LIN {X -0.145,Y -338.267,Z 1435.514,A 0.000,B 0.000,C 90.000,E1 272.579} C_DIS
LIN {X 0.126,Y -330.256,Z 1435.514,A 0.000,B 0.000,C 90.000,E1 272.407} C_DIS
LIN {X -0.143,Y -321.454,Z 1435.513,A 0.000,B 0.000,C 90.000,E1 272.350} C_DIS
LIN {X 0.117,Y -311.305,Z 1435.513,A 0.000,B 0.000,C 90.000,E1 272.236} C_DIS
LIN {X 0.012,Y -305.881,Z 1435.512,A 0.000,B 0.000,C 90.000,E1 272.236} C_DIS
LIN {X -0.024,Y -181.226,Z 1435.512,A 0.000,B 0.000,C 90.000,E1 272.236} C_DIS
LIN {X 0.021,Y -181.579,Z 1435.501,A 0.000,B 0.000,C 90.000,E1 270.172} C_DIS
LIN {X 0.010,Y -180.886,Z 1435.473,A 0.000,B 0.000,C 90.000,E1 265.122} C_DIS
LIN {X 0.070,Y -179.008,Z 1435.445,A 0.000,B 0.000,C 90.000,E1 260.038} C_DIS
LIN {X -0.012,Y -178.617,Z 1435.440,A 0.000,B 0.000,C 90.000,E1 259.218} C_DIS
LIN {X 0.056,Y -175.669,Z 1435.412,A 0.000,B 0.000,C 90.000,E1 254.102} C_DIS
LIN {X 0.061,Y -172.386,Z 1435.388,A 0.000,B 0.000,C 90.000,E1 249.826} C_DIS
LIN {X 0.075,Y -171.187,Z 1435.379,A 0.000,B 0.000,C 90.000,E1 248.103} C_DIS
LIN {X -0.032,Y -167.479,Z 1435.354,A 0.000,B 0.000,C 90.000,E1 243.819} C_DIS
LIN {X -0.025,Y -166.875,Z 1435.350,A 0.000,B 0.000,C 90.000,E1 242.948} C_DIS
LIN {X -0.032,Y -162.180,Z 1435.321,A 0.000,B 0.000,C 90.000,E1 237.709} C_DIS
LIN {X 0.025,Y -160.746,Z 1435.311,A 0.000,B 0.000,C 90.000,E1 235.928} C_DIS
LIN {X 0.003,Y -157.546,Z 1435.291,A 0.000,B 0.000,C 90.000,E1 232.396} C_DIS
LIN {X -0.058,Y -155.574,Z 1435.276,A 0.000,B 0.000,C 90.000,E1 229.747} C_DIS
LIN {X -0.006,Y -151.860,Z 1435.251,A 0.000,B 0.000,C 90.000,E1 225.243} C_DIS
LIN {X 0.007,Y -150.083,Z 1435.236,A 0.000,B 0.000,C 90.000,E1 222.528} C_DIS
LIN {X 0.041,Y -146.886,Z 1435.211,A 0.000,B 0.000,C 90.000,E1 217.971} C_DIS
LIN {X 0.030,Y -145.473,Z 1435.196,A 0.000,B 0.000,C 90.000,E1 215.231} C_DIS
LIN {X -0.053,Y -142.884,Z 1435.170,A 0.000,B 0.000,C 90.000,E1 210.669} C_DIS
LIN {X 0.004,Y -141.503,Z 1435.150,A 0.000,B 0.000,C 90.000,E1 206.950} C_DIS
LIN {X 0.053,Y -139.389,Z 1435.114,A 0.000,B 0.000,C 90.000,E1 200.429} C_DIS
LIN {X -0.027,Y -139.096,Z 1435.103,A 0.000,B 0.000,C 90.000,E1 198.598} C_DIS
LIN {X -0.035,Y -138.353,Z 1435.057,A 0.000,B 0.000,C 90.000,E1 190.197} C_DIS
LIN {X -0.043,Y -139.516,Z 1435.005,A 0.000,B 0.000,C 90.000,E1 180.859} C_DIS
LIN {X 0.038,Y -141.171,Z 1434.974,A 0.000,B 0.000,C 90.000,E1 175.241} C_DIS
LIN {X 0.009,Y -142.550,Z 1434.958,A 0.000,B 0.000,C 90.000,E1 172.470} C_DIS
LIN {X -0.065,Y -144.826,Z 1434.932,A 0.000,B 0.000,C 90.000,E1 167.881} C_DIS
LIN {X 0.063,Y -147.449,Z 1434.912,A 0.000,B 0.000,C 90.000,E1 164.157} C_DIS
LIN {X -0.050,Y -150.030,Z 1434.892,A 0.000,B 0.000,C 90.000,E1 160.550} C_DIS
LIN {X -0.044,Y -153.367,Z 1434.872,A 0.000,B 0.000,C 90.000,E1 156.922} C_DIS
LIN {X 0.005,Y -155.901,Z 1434.857,A 0.000,B 0.000,C 90.000,E1 154.204} C_DIS
LIN {X -0.019,Y -159.761,Z 1434.837,A 0.000,B 0.000,C 90.000,E1 150.639} C_DIS
LIN {X -0.032,Y -162.001,Z 1434.827,A 0.000,B 0.000,C 90.000,E1 148.869} C_DIS
LIN {X -0.013,Y -166.194,Z 1434.807,A 0.000,B 0.000,C 90.000,E1 145.341} C_DIS
LIN {X 0.085,Y -171.208,Z 1434.788,A 0.000,B 0.000,C 90.000,E1 141.823} C_DIS
LIN {X 0.009,Y -176.093,Z 1434.769,A 0.000,B 0.000,C 90.000,E1 138.405} C_DIS
LIN {X 0.000,Y -180.354,Z 1434.755,A 0.000,B 0.000,C 90.000,E1 135.850} C_DIS
LIN {X 0.104,Y -185.763,Z 1434.736,A 0.000,B 0.000,C 90.000,E1 132.447} C_DIS
LIN {X 0.037,Y -190.377,Z 1434.722,A 0.000,B 0.000,C 90.000,E1 129.967} C_DIS
LIN {X -0.063,Y -197.702,Z 1434.699,A 0.000,B 0.000,C 90.000,E1 125.884} C_DIS
LIN {X -0.012,Y -200.248,Z 1434.692,A 0.000,B 0.000,C 90.000,E1 124.612} C_DIS
LIN {X -0.078,Y -312.029,Z 1434.692,A 0.000,B 0.000,C 90.000,E1 124.612} C_DIS
LIN {X 0.044,Y -317.244,Z 1434.691,A 0.000,B 0.000,C 90.000,E1 124.405} C_DIS
LIN {X -0.034,Y -319.611,Z 1434.690,A 0.000,B 0.000,C 90.000,E1 124.246} C_DIS
LIN {X 0.116,Y -323.459,Z 1434.688,A 0.000,B 0.000,C 90.000,E1 123.785} C_DIS
LIN {X 0.010,Y -325.330,Z 1434.686,A 0.000,B 0.000,C 90.000,E1 123.499} C_DIS
LIN {X -0.099,Y -326.795,Z 1434.684,A 0.000,B 0.000,C 90.000,E1 123.214} C_DIS
LIN {X 0.023,Y -339.885,Z 1434.665,A 0.000,B 0.000,C 90.000,E1 119.745} C_DIS
LIN {X -0.091,Y -352.024,Z 1434.650,A 0.000,B 0.000,C 90.000,E1 117.001} C_DIS
LIN {X 0.137,Y -365.628,Z 1434.635,A 0.000,B 0.000,C 90.000,E1 114.259} C_DIS
LIN {X 0.193,Y -379.053,Z 1434.622,A 0.000,B 0.000,C 90.000,E1 111.897} C_DIS
LIN {X -0.052,Y -393.825,Z 1434.609,A 0.000,B 0.000,C 90.000,E1 109.631} C_DIS
LIN {X -0.205,Y -410.046,Z 1434.597,A 0.000,B 0.000,C 90.000,E1 107.402} C_DIS
LIN {X -0.078,Y -427.833,Z 1434.584,A 0.000,B 0.000,C 90.000,E1 105.190} C_DIS
LIN {X -0.073,Y -447.205,Z 1434.573,A 0.000,B 0.000,C 90.000,E1 103.063} C_DIS
LIN {X 0.056,Y -467.384,Z 1434.562,A 0.000,B 0.000,C 90.000,E1 101.074} C_DIS
LIN {X -0.132,Y -485.488,Z 1434.553,A 0.000,B 0.000,C 90.000,E1 99.500} C_DIS
LIN {X 0.022,Y -487.773,Z 1434.552,A 0.000,B 0.000,C 90.000,E1 99.265} C_DIS
LIN {X 0.176,Y -489.501,Z 1434.550,A 0.000,B 0.000,C 90.000,E1 99.029} C_DIS
LIN {X -0.002,Y -490.998,Z 1434.549,A 0.000,B 0.000,C 90.000,E1 98.803} C_DIS
LIN {X -0.103,Y -492.112,Z 1434.547,A 0.000,B 0.000,C 90.000,E1 98.568} C_DIS
LIN {X 0.124,Y -493.421,Z 1434.545,A 0.000,B 0.000,C 90.000,E1 98.049} C_DIS
LIN {X -0.129,Y -493.693,Z 1434.542,A 0.000,B 0.000,C 90.000,E1 97.587} C_DIS
LIN {X 0.117,Y -492.973,Z 1434.539,A 0.000,B 0.000,C 90.000,E1 97.068} C_DIS
LIN {X -0.125,Y -491.140,Z 1434.537,A 0.000,B 0.000,C 90.000,E1 96.606} C_DIS
LIN {X -0.221,Y -489.699,Z 1434.535,A 0.000,B 0.000,C 90.000,E1 96.372} C_DIS
LIN {X 0.050,Y -476.478,Z 1434.524,A 0.000,B 0.000,C 90.000,E1 94.359} C_DIS
LIN {X 0.126,Y -468.748,Z 1434.517,A 0.000,B 0.000,C 90.000,E1 93.094} C_DIS
LIN {X 0.040,Y -460.487,Z 1434.510,A 0.000,B 0.000,C 90.000,E1 91.835} C_DIS
LIN {X 0.052,Y -446.989,Z 1434.499,A 0.000,B 0.000,C 90.000,E1 89.771} C_DIS
LIN {X 0.071,Y -430.842,Z 1434.484,A 0.000,B 0.000,C 90.000,E1 87.135} C_DIS
LIN {X 0.169,Y -419.506,Z 1434.474,A 0.000,B 0.000,C 90.000,E1 85.241} C_DIS
LIN {X -0.006,Y -409.767,Z 1434.465,A 0.000,B 0.000,C 90.000,E1 83.628} C_DIS
LIN {X 0.192,Y -398.368,Z 1434.454,A 0.000,B 0.000,C 90.000,E1 81.659} C_DIS
LIN {X 0.153,Y -386.689,Z 1434.443,A 0.000,B 0.000,C 90.000,E1 79.690} C_DIS
LIN {X 0.023,Y -371.879,Z 1434.428,A 0.000,B 0.000,C 90.000,E1 77.117} C_DIS
LIN {X 0.103,Y -360.596,Z 1434.417,A 0.000,B 0.000,C 90.000,E1 75.046} C_DIS
LIN {X 0.006,Y -350.893,Z 1434.407,A 0.000,B 0.000,C 90.000,E1 73.268} C_DIS
LIN {X -0.058,Y -339.370,Z 1434.395,A 0.000,B 0.000,C 90.000,E1 71.148} C_DIS
LIN {X 0.075,Y -327.939,Z 1434.383,A 0.000,B 0.000,C 90.000,E1 68.954} C_DIS
LIN {X 0.059,Y -313.709,Z 1434.367,A 0.000,B 0.000,C 90.000,E1 66.102} C_DIS
LIN {X 0.019,Y -301.931,Z 1434.353,A 0.000,B 0.000,C 90.000,E1 63.512} C_DIS
LIN {X -0.058,Y -288.636,Z 1434.334,A 0.000,B 0.000,C 90.000,E1 60.205} C_DIS
LIN {X 0.031,Y -276.569,Z 1434.316,A 0.000,B 0.000,C 90.000,E1 56.786} C_DIS
LIN {X -0.168,Y -266.379,Z 1434.298,A 0.000,B 0.000,C 90.000,E1 53.703} C_DIS
LIN {X 0.058,Y -255.745,Z 1434.278,A 0.000,B 0.000,C 90.000,E1 50.114} C_DIS
LIN {X -0.098,Y -246.028,Z 1434.258,A 0.000,B 0.000,C 90.000,E1 46.539} C_DIS
LIN {X -0.060,Y -237.200,Z 1434.238,A 0.000,B 0.000,C 90.000,E1 42.852} C_DIS
LIN {X -0.091,Y -229.202,Z 1434.217,A 0.000,B 0.000,C 90.000,E1 39.116} C_DIS
LIN {X -0.089,Y -222.060,Z 1434.196,A 0.000,B 0.000,C 90.000,E1 35.311} C_DIS
LIN {X 0.043,Y -215.774,Z 1434.175,A 0.000,B 0.000,C 90.000,E1 31.416} C_DIS
LIN {X 0.010,Y -210.245,Z 1434.153,A 0.000,B 0.000,C 90.000,E1 27.513} C_DIS
LIN {X -0.029,Y -205.570,Z 1434.131,A 0.000,B 0.000,C 90.000,E1 23.567} C_DIS
LIN {X -0.066,Y -201.069,Z 1434.104,A 0.000,B 0.000,C 90.000,E1 18.779} C_DIS
LIN {X -0.076,Y -197.698,Z 1434.077,A 0.000,B 0.000,C 90.000,E1 13.939} C_DIS
LIN {X 0.037,Y -195.219,Z 1434.050,A 0.000,B 0.000,C 90.000,E1 9.029} C_DIS
LIN {X 0.028,Y -193.585,Z 1434.023,A 0.000,B 0.000,C 90.000,E1 4.131} C_DIS
LIN {X 0.095,Y -192.597,Z 1433.993,A 0.000,B 0.000,C 90.000,E1 358.682} C_DIS
LIN {X -0.049,Y -192.475,Z 1433.965,A 0.000,B 0.000,C 90.000,E1 353.799} C_DIS
LIN {X -0.037,Y -193.142,Z 1433.934,A 0.000,B 0.000,C 90.000,E1 348.049} C_DIS
LIN {X -0.074,Y -195.715,Z 1433.897,A 0.000,B 0.000,C 90.000,E1 341.511} C_DIS
LIN {X -0.024,Y -199.234,Z 1433.870,A 0.000,B 0.000,C 90.000,E1 336.613} C_DIS
LIN {X 0.017,Y -203.361,Z 1433.848,A 0.000,B 0.000,C 90.000,E1 332.564} C_DIS
LIN {X -0.051,Y -208.601,Z 1433.825,A 0.000,B 0.000,C 90.000,E1 328.584} C_DIS
LIN {X 0.060,Y -213.728,Z 1433.808,A 0.000,B 0.000,C 90.000,E1 325.388} C_DIS
LIN {X 0.014,Y -219.879,Z 1433.790,A 0.000,B 0.000,C 90.000,E1 322.271} C_DIS
LIN {X 0.041,Y -226.992,Z 1433.773,A 0.000,B 0.000,C 90.000,E1 319.175} C_DIS
LIN {X 0.005,Y -236.100,Z 1433.754,A 0.000,B 0.000,C 90.000,E1 315.769} C_DIS
LIN {X 0.090,Y -245.170,Z 1433.738,A 0.000,B 0.000,C 90.000,E1 312.771} C_DIS
LIN {X 0.108,Y -256.587,Z 1433.719,A 0.000,B 0.000,C 90.000,E1 309.483} C_DIS
LIN {X -0.062,Y -267.968,Z 1433.704,A 0.000,B 0.000,C 90.000,E1 306.664} C_DIS
LIN {X 0.025,Y -279.257,Z 1433.690,A 0.000,B 0.000,C 90.000,E1 304.199} C_DIS
LIN {X -0.015,Y -286.345,Z 1433.682,A 0.000,B 0.000,C 90.000,E1 302.832} C_DIS
LIN {X 0.036,Y -294.207,Z 1433.675,A 0.000,B 0.000,C 90.000,E1 301.465} C_DIS
LIN {X 0.043,Y -304.988,Z 1433.666,A 0.000,B 0.000,C 90.000,E1 299.795} C_DIS
LIN {X 0.023,Y -314.696,Z 1433.658,A 0.000,B 0.000,C 90.000,E1 298.487} C_DIS
LIN {X 0.044,Y -327.610,Z 1433.650,A 0.000,B 0.000,C 90.000,E1 296.950} C_DIS
LIN {X -0.026,Y -349.254,Z 1433.637,A 0.000,B 0.000,C 90.000,E1 294.695} C_DIS
LIN {X -0.169,Y -362.739,Z 1433.630,A 0.000,B 0.000,C 90.000,E1 293.334} C_DIS
LIN {X -0.059,Y -373.323,Z 1433.623,A 0.000,B 0.000,C 90.000,E1 292.206} C_DIS
LIN {X -0.032,Y -386.257,Z 1433.615,A 0.000,B 0.000,C 90.000,E1 290.791} C_DIS
LIN {X 0.149,Y -396.447,Z 1433.609,A 0.000,B 0.000,C 90.000,E1 289.631} C_DIS
LIN {X 0.159,Y -411.444,Z 1433.600,A 0.000,B 0.000,C 90.000,E1 287.946} C_DIS
LIN {X -0.072,Y -418.826,Z 1433.595,A 0.000,B 0.000,C 90.000,E1 287.149} C_DIS
LIN {X 0.042,Y -425.619,Z 1433.591,A 0.000,B 0.000,C 90.000,E1 286.315} C_DIS
LIN {X -0.062,Y -429.691,Z 1433.588,A 0.000,B 0.000,C 90.000,E1 285.788} C_DIS
LIN {X -0.023,Y -433.376,Z 1433.585,A 0.000,B 0.000,C 90.000,E1 285.245} C_DIS
LIN {X 0.114,Y -438.048,Z 1433.580,A 0.000,B 0.000,C 90.000,E1 284.426} C_DIS
LIN {X -0.015,Y -441.908,Z 1433.576,A 0.000,B 0.000,C 90.000,E1 283.647} C_DIS
LIN {X 0.210,Y -445.060,Z 1433.571,A 0.000,B 0.000,C 90.000,E1 282.827} C_DIS
LIN {X -0.207,Y -446.761,Z 1433.568,A 0.000,B 0.000,C 90.000,E1 282.355} C_DIS
LIN {X -0.178,Y -448.130,Z 1433.566,A 0.000,B 0.000,C 90.000,E1 281.827} C_DIS
LIN {X -0.141,Y -449.139,Z 1433.563,A 0.000,B 0.000,C 90.000,E1 281.299} C_DIS
LIN {X -0.180,Y -449.709,Z 1433.560,A 0.000,B 0.000,C 90.000,E1 280.782} C_DIS
LIN {X -0.128,Y -449.834,Z 1433.557,A 0.000,B 0.000,C 90.000,E1 280.254} C_DIS
LIN {X -0.076,Y -449.495,Z 1433.554,A 0.000,B 0.000,C 90.000,E1 279.726} C_DIS
LIN {X -0.098,Y -448.642,Z 1433.551,A 0.000,B 0.000,C 90.000,E1 279.208} C_DIS
LIN {X -0.050,Y -447.164,Z 1433.548,A 0.000,B 0.000,C 90.000,E1 278.681} C_DIS
LIN {X -0.077,Y -445.065,Z 1433.545,A 0.000,B 0.000,C 90.000,E1 278.163} C_DIS
LIN {X 0.157,Y -443.775,Z 1433.544,A 0.000,B 0.000,C 90.000,E1 277.871} C_DIS
LIN {X 0.113,Y -440.529,Z 1433.541,A 0.000,B 0.000,C 90.000,E1 277.352} C_DIS
LIN {X -0.158,Y -438.557,Z 1433.539,A 0.000,B 0.000,C 90.000,E1 277.125} C_DIS
LIN {X -0.223,Y -433.757,Z 1433.536,A 0.000,B 0.000,C 90.000,E1 276.606} C_DIS
LIN {X 0.144,Y -427.709,Z 1433.534,A 0.000,B 0.000,C 90.000,E1 276.030} C_DIS
LIN {X -0.192,Y -421.451,Z 1433.531,A 0.000,B 0.000,C 90.000,E1 275.625} C_DIS
LIN {X -0.102,Y -414.920,Z 1433.529,A 0.000,B 0.000,C 90.000,E1 275.220} C_DIS
LIN {X 0.100,Y -405.272,Z 1433.526,A 0.000,B 0.000,C 90.000,E1 274.702} C_DIS
LIN {X 0.072,Y -398.765,Z 1433.525,A 0.000,B 0.000,C 90.000,E1 274.416} C_DIS
LIN {X 0.148,Y -385.981,Z 1433.522,A 0.000,B 0.000,C 90.000,E1 273.898} C_DIS
LIN {X 0.082,Y -373.099,Z 1433.519,A 0.000,B 0.000,C 90.000,E1 273.440} C_DIS
LIN {X -0.154,Y -363.120,Z 1433.517,A 0.000,B 0.000,C 90.000,E1 273.151} C_DIS
LIN {X 0.060,Y -356.360,Z 1433.516,A 0.000,B 0.000,C 90.000,E1 272.922} C_DIS
LIN {X -0.102,Y -345.391,Z 1433.515,A 0.000,B 0.000,C 90.000,E1 272.694} C_DIS
LIN {X 0.077,Y -338.067,Z 1433.514,A 0.000,B 0.000,C 90.000,E1 272.522} C_DIS
LIN {X 0.032,Y -329.934,Z 1433.513,A 0.000,B 0.000,C 90.000,E1 272.407} C_DIS
LIN {X -0.033,Y -317.499,Z 1433.513,A 0.000,B 0.000,C 90.000,E1 272.293} C_DIS
LIN {X 0.007,Y -306.470,Z 1433.512,A 0.000,B 0.000,C 90.000,E1 272.236} C_DIS
LIN {X -0.024,Y -181.226,Z 1433.512,A 0.000,B 0.000,C 90.000,E1 272.236} C_DIS
LIN {X -0.023,Y -181.564,Z 1433.503,A 0.000,B 0.000,C 90.000,E1 270.516} C_DIS
LIN {X -0.034,Y -181.121,Z 1433.489,A 0.000,B 0.000,C 90.000,E1 267.993} C_DIS
LIN {X -0.045,Y -180.907,Z 1433.475,A 0.000,B 0.000,C 90.000,E1 265.469} C_DIS
LIN {X 0.012,Y -180.730,Z 1433.470,A 0.000,B 0.000,C 90.000,E1 264.609} C_DIS
LIN {X -0.066,Y -178.819,Z 1433.442,A 0.000,B 0.000,C 90.000,E1 259.567} C_DIS
LIN {X 0.015,Y -175.864,Z 1433.414,A 0.000,B 0.000,C 90.000,E1 254.448} C_DIS
LIN {X 0.064,Y -173.831,Z 1433.399,A 0.000,B 0.000,C 90.000,E1 251.873} C_DIS
LIN {X -0.001,Y -171.499,Z 1433.380,A 0.000,B 0.000,C 90.000,E1 248.465} C_DIS
LIN {X -0.014,Y -167.727,Z 1433.356,A 0.000,B 0.000,C 90.000,E1 244.152} C_DIS
LIN {X 0.002,Y -166.422,Z 1433.347,A 0.000,B 0.000,C 90.000,E1 242.410} C_DIS
LIN {X 0.000,Y -163.143,Z 1433.327,A 0.000,B 0.000,C 90.000,E1 238.918} C_DIS
LIN {X -0.034,Y -161.098,Z 1433.313,A 0.000,B 0.000,C 90.000,E1 236.294} C_DIS
LIN {X -0.050,Y -157.826,Z 1433.293,A 0.000,B 0.000,C 90.000,E1 232.763} C_DIS
LIN {X 0.013,Y -155.860,Z 1433.278,A 0.000,B 0.000,C 90.000,E1 230.070} C_DIS
LIN {X 0.069,Y -152.109,Z 1433.253,A 0.000,B 0.000,C 90.000,E1 225.567} C_DIS
LIN {X -0.024,Y -150.360,Z 1433.238,A 0.000,B 0.000,C 90.000,E1 222.894} C_DIS
LIN {X 0.016,Y -147.095,Z 1433.213,A 0.000,B 0.000,C 90.000,E1 218.338} C_DIS
LIN {X 0.011,Y -145.665,Z 1433.198,A 0.000,B 0.000,C 90.000,E1 215.598} C_DIS
LIN {X 0.013,Y -143.048,Z 1433.172,A 0.000,B 0.000,C 90.000,E1 211.003} C_DIS
LIN {X 0.014,Y -141.671,Z 1433.152,A 0.000,B 0.000,C 90.000,E1 207.308} C_DIS
LIN {X 0.058,Y -139.452,Z 1433.116,A 0.000,B 0.000,C 90.000,E1 200.791} C_DIS
LIN {X -0.021,Y -139.186,Z 1433.105,A 0.000,B 0.000,C 90.000,E1 198.960} C_DIS
LIN {X 0.002,Y -138.322,Z 1433.053,A 0.000,B 0.000,C 90.000,E1 189.613} C_DIS
LIN {X 0.009,Y -139.460,Z 1433.007,A 0.000,B 0.000,C 90.000,E1 181.203} C_DIS
LIN {X -0.051,Y -141.016,Z 1432.976,A 0.000,B 0.000,C 90.000,E1 175.641} C_DIS
LIN {X 0.040,Y -142.770,Z 1432.955,A 0.000,B 0.000,C 90.000,E1 171.894} C_DIS
LIN {X -0.005,Y -145.180,Z 1432.929,A 0.000,B 0.000,C 90.000,E1 167.297} C_DIS
LIN {X 0.028,Y -147.802,Z 1432.909,A 0.000,B 0.000,C 90.000,E1 163.614} C_DIS
LIN {X -0.077,Y -150.488,Z 1432.889,A 0.000,B 0.000,C 90.000,E1 160.007} C_DIS
LIN {X -0.004,Y -153.943,Z 1432.869,A 0.000,B 0.000,C 90.000,E1 156.357} C_DIS
LIN {X 0.059,Y -157.354,Z 1432.849,A 0.000,B 0.000,C 90.000,E1 152.743} C_DIS
LIN {X 0.003,Y -161.551,Z 1432.829,A 0.000,B 0.000,C 90.000,E1 149.203} C_DIS
LIN {X 0.014,Y -165.749,Z 1432.809,A 0.000,B 0.000,C 90.000,E1 145.674} C_DIS
LIN {X 0.002,Y -170.703,Z 1432.790,A 0.000,B 0.000,C 90.000,E1 142.190} C_DIS
LIN {X -0.087,Y -175.576,Z 1432.771,A 0.000,B 0.000,C 90.000,E1 138.771} C_DIS
LIN {X 0.032,Y -181.194,Z 1432.752,A 0.000,B 0.000,C 90.000,E1 135.324} C_DIS
LIN {X 0.026,Y -186.655,Z 1432.733,A 0.000,B 0.000,C 90.000,E1 131.962} C_DIS
LIN {X -0.030,Y -191.260,Z 1432.719,A 0.000,B 0.000,C 90.000,E1 129.483} C_DIS
LIN {X 0.050,Y -197.081,Z 1432.701,A 0.000,B 0.000,C 90.000,E1 126.171} C_DIS
LIN {X 0.063,Y -200.204,Z 1432.692,A 0.000,B 0.000,C 90.000,E1 124.612} C_DIS
LIN {X 0.063,Y -311.776,Z 1432.692,A 0.000,B 0.000,C 90.000,E1 124.612} C_DIS
LIN {X 0.137,Y -314.663,Z 1432.692,A 0.000,B 0.000,C 90.000,E1 124.532} C_DIS
LIN {X -0.170,Y -318.101,Z 1432.691,A 0.000,B 0.000,C 90.000,E1 124.405} C_DIS
LIN {X 0.050,Y -321.655,Z 1432.689,A 0.000,B 0.000,C 90.000,E1 124.040} C_DIS
LIN {X 0.153,Y -325.220,Z 1432.686,A 0.000,B 0.000,C 90.000,E1 123.499} C_DIS
LIN {X -0.032,Y -326.743,Z 1432.684,A 0.000,B 0.000,C 90.000,E1 123.214} C_DIS
LIN {X 0.079,Y -339.825,Z 1432.665,A 0.000,B 0.000,C 90.000,E1 119.745} C_DIS
LIN {X -0.030,Y -351.955,Z 1432.650,A 0.000,B 0.000,C 90.000,E1 117.001} C_DIS
LIN {X 0.042,Y -365.558,Z 1432.635,A 0.000,B 0.000,C 90.000,E1 114.283} C_DIS
LIN {X -0.102,Y -378.978,Z 1432.622,A 0.000,B 0.000,C 90.000,E1 111.950} C_DIS
LIN {X 0.003,Y -393.744,Z 1432.609,A 0.000,B 0.000,C 90.000,E1 109.631} C_DIS
LIN {X -0.149,Y -409.961,Z 1432.597,A 0.000,B 0.000,C 90.000,E1 107.402} C_DIS
LIN {X -0.022,Y -427.741,Z 1432.584,A 0.000,B 0.000,C 90.000,E1 105.190} C_DIS
LIN {X -0.029,Y -447.125,Z 1432.573,A 0.000,B 0.000,C 90.000,E1 103.063} C_DIS
LIN {X 0.097,Y -467.302,Z 1432.562,A 0.000,B 0.000,C 90.000,E1 101.074} C_DIS
LIN {X -0.073,Y -485.377,Z 1432.553,A 0.000,B 0.000,C 90.000,E1 99.500} C_DIS
LIN {X 0.060,Y -487.677,Z 1432.552,A 0.000,B 0.000,C 90.000,E1 99.265} C_DIS
LIN {X 0.043,Y -489.534,Z 1432.550,A 0.000,B 0.000,C 90.000,E1 99.029} C_DIS
LIN {X -0.049,Y -490.939,Z 1432.549,A 0.000,B 0.000,C 90.000,E1 98.803} C_DIS
LIN {X 0.242,Y -492.810,Z 1432.546,A 0.000,B 0.000,C 90.000,E1 98.276} C_DIS
LIN {X -0.019,Y -493.556,Z 1432.543,A 0.000,B 0.000,C 90.000,E1 97.814} C_DIS
LIN {X 0.219,Y -493.308,Z 1432.541,A 0.000,B 0.000,C 90.000,E1 97.296} C_DIS
LIN {X -0.027,Y -492.029,Z 1432.538,A 0.000,B 0.000,C 90.000,E1 96.834} C_DIS
LIN {X -0.178,Y -490.940,Z 1432.537,A 0.000,B 0.000,C 90.000,E1 96.606} C_DIS
LIN {X 0.060,Y -487.770,Z 1432.534,A 0.000,B 0.000,C 90.000,E1 96.087} C_DIS
LIN {X -0.006,Y -476.274,Z 1432.524,A 0.000,B 0.000,C 90.000,E1 94.359} C_DIS
LIN {X 0.065,Y -468.519,Z 1432.517,A 0.000,B 0.000,C 90.000,E1 93.094} C_DIS
LIN {X -0.020,Y -460.231,Z 1432.510,A 0.000,B 0.000,C 90.000,E1 91.835} C_DIS
LIN {X -0.011,Y -446.743,Z 1432.499,A 0.000,B 0.000,C 90.000,E1 89.771} C_DIS
LIN {X 0.004,Y -430.684,Z 1432.484,A 0.000,B 0.000,C 90.000,E1 87.135} C_DIS
LIN {X 0.095,Y -419.356,Z 1432.474,A 0.000,B 0.000,C 90.000,E1 85.241} C_DIS
LIN {X -0.080,Y -409.634,Z 1432.464,A 0.000,B 0.000,C 90.000,E1 83.628} C_DIS
LIN {X 0.122,Y -398.275,Z 1432.454,A 0.000,B 0.000,C 90.000,E1 81.659} C_DIS
LIN {X 0.078,Y -386.602,Z 1432.443,A 0.000,B 0.000,C 90.000,E1 79.690} C_DIS
LIN {X -0.055,Y -373.439,Z 1432.430,A 0.000,B 0.000,C 90.000,E1 77.409} C_DIS
LIN {X 0.063,Y -362.148,Z 1432.419,A 0.000,B 0.000,C 90.000,E1 75.338} C_DIS
LIN {X -0.002,Y -352.446,Z 1432.409,A 0.000,B 0.000,C 90.000,E1 73.559} C_DIS
LIN {X -0.146,Y -342.594,Z 1432.399,A 0.000,B 0.000,C 90.000,E1 71.764} C_DIS
LIN {X 0.049,Y -331.119,Z 1432.387,A 0.000,B 0.000,C 90.000,E1 69.571} C_DIS
LIN {X -0.001,Y -316.706,Z 1432.371,A 0.000,B 0.000,C 90.000,E1 66.741} C_DIS
LIN {X 0.058,Y -303.244,Z 1432.355,A 0.000,B 0.000,C 90.000,E1 63.819} C_DIS
LIN {X 0.027,Y -289.813,Z 1432.336,A 0.000,B 0.000,C 90.000,E1 60.511} C_DIS
LIN {X 0.012,Y -277.679,Z 1432.317,A 0.000,B 0.000,C 90.000,E1 57.120} C_DIS
LIN {X 0.064,Y -267.490,Z 1432.300,A 0.000,B 0.000,C 90.000,E1 53.989} C_DIS
LIN {X -0.053,Y -256.772,Z 1432.280,A 0.000,B 0.000,C 90.000,E1 50.481} C_DIS
LIN {X 0.012,Y -247.002,Z 1432.260,A 0.000,B 0.000,C 90.000,E1 46.863} C_DIS
LIN {X 0.076,Y -238.115,Z 1432.240,A 0.000,B 0.000,C 90.000,E1 43.176} C_DIS
LIN {X 0.074,Y -230.059,Z 1432.219,A 0.000,B 0.000,C 90.000,E1 39.439} C_DIS
LIN {X 0.055,Y -222.842,Z 1432.198,A 0.000,B 0.000,C 90.000,E1 35.644} C_DIS
LIN {X 0.018,Y -216.498,Z 1432.177,A 0.000,B 0.000,C 90.000,E1 31.799} C_DIS
LIN {X 0.003,Y -210.891,Z 1432.155,A 0.000,B 0.000,C 90.000,E1 27.897} C_DIS
LIN {X -0.015,Y -206.166,Z 1432.133,A 0.000,B 0.000,C 90.000,E1 23.951} C_DIS
LIN {X 0.046,Y -201.622,Z 1432.106,A 0.000,B 0.000,C 90.000,E1 19.141} C_DIS
LIN {X 0.057,Y -198.187,Z 1432.080,A 0.000,B 0.000,C 90.000,E1 14.300} C_DIS
LIN {X 0.021,Y -195.344,Z 1432.048,A 0.000,B 0.000,C 90.000,E1 8.624} C_DIS
LIN {X 0.061,Y -194.008,Z 1432.025,A 0.000,B 0.000,C 90.000,E1 4.531} C_DIS
LIN {X -0.035,Y -192.978,Z 1431.997,A 0.000,B 0.000,C 90.000,E1 359.542} C_DIS
LIN {X -0.037,Y -192.761,Z 1431.965,A 0.000,B 0.000,C 90.000,E1 353.799} C_DIS
LIN {X -0.014,Y -193.412,Z 1431.934,A 0.000,B 0.000,C 90.000,E1 348.049} C_DIS
LIN {X -0.038,Y -195.940,Z 1431.897,A 0.000,B 0.000,C 90.000,E1 341.511} C_DIS
LIN {X 0.021,Y -199.430,Z 1431.870,A 0.000,B 0.000,C 90.000,E1 336.613} C_DIS
LIN {X -0.111,Y -203.566,Z 1431.848,A 0.000,B 0.000,C 90.000,E1 332.615} C_DIS
LIN {X 0.009,Y -208.787,Z 1431.825,A 0.000,B 0.000,C 90.000,E1 328.584} C_DIS
LIN {X 0.127,Y -213.917,Z 1431.808,A 0.000,B 0.000,C 90.000,E1 325.388} C_DIS
LIN {X 0.086,Y -220.063,Z 1431.791,A 0.000,B 0.000,C 90.000,E1 322.271} C_DIS
LIN {X -0.051,Y -227.163,Z 1431.773,A 0.000,B 0.000,C 90.000,E1 319.218} C_DIS
LIN {X -0.082,Y -236.262,Z 1431.754,A 0.000,B 0.000,C 90.000,E1 315.810} C_DIS
LIN {X -0.013,Y -246.529,Z 1431.736,A 0.000,B 0.000,C 90.000,E1 312.447} C_DIS
LIN {X -0.126,Y -258.086,Z 1431.718,A 0.000,B 0.000,C 90.000,E1 309.197} C_DIS
LIN {X 0.113,Y -269.596,Z 1431.702,A 0.000,B 0.000,C 90.000,E1 306.297} C_DIS
LIN {X 0.079,Y -281.049,Z 1431.688,A 0.000,B 0.000,C 90.000,E1 303.865} C_DIS
LIN {X 0.066,Y -288.301,Z 1431.681,A 0.000,B 0.000,C 90.000,E1 302.498} C_DIS
LIN {X 0.144,Y -300.572,Z 1431.669,A 0.000,B 0.000,C 90.000,E1 300.463} C_DIS
LIN {X 0.072,Y -309.738,Z 1431.662,A 0.000,B 0.000,C 90.000,E1 299.155} C_DIS
LIN {X -0.137,Y -322.067,Z 1431.653,A 0.000,B 0.000,C 90.000,E1 297.641} C_DIS
LIN {X 0.065,Y -332.776,Z 1431.647,A 0.000,B 0.000,C 90.000,E1 296.411} C_DIS
LIN {X -0.075,Y -351.818,Z 1431.636,A 0.000,B 0.000,C 90.000,E1 294.463} C_DIS
LIN {X -0.057,Y -365.223,Z 1431.628,A 0.000,B 0.000,C 90.000,E1 293.078} C_DIS
LIN {X -0.109,Y -375.716,Z 1431.622,A 0.000,B 0.000,C 90.000,E1 291.972} C_DIS
LIN {X -0.127,Y -388.630,Z 1431.614,A 0.000,B 0.000,C 90.000,E1 290.556} C_DIS
LIN {X -0.086,Y -401.158,Z 1431.606,A 0.000,B 0.000,C 90.000,E1 289.141} C_DIS
LIN {X 0.044,Y -416.135,Z 1431.597,A 0.000,B 0.000,C 90.000,E1 287.457} C_DIS
LIN {X 0.130,Y -423.196,Z 1431.592,A 0.000,B 0.000,C 90.000,E1 286.622} C_DIS
LIN {X -0.120,Y -429.517,Z 1431.588,A 0.000,B 0.000,C 90.000,E1 285.843} C_DIS
LIN {X 0.091,Y -434.908,Z 1431.583,A 0.000,B 0.000,C 90.000,E1 285.009} C_DIS
LIN {X -0.174,Y -439.369,Z 1431.579,A 0.000,B 0.000,C 90.000,E1 284.245} C_DIS
LIN {X 0.129,Y -443.030,Z 1431.575,A 0.000,B 0.000,C 90.000,E1 283.411} C_DIS
LIN {X 0.141,Y -445.110,Z 1431.572,A 0.000,B 0.000,C 90.000,E1 282.883} C_DIS
LIN {X 0.164,Y -446.862,Z 1431.569,A 0.000,B 0.000,C 90.000,E1 282.355} C_DIS
LIN {X 0.194,Y -448.267,Z 1431.566,A 0.000,B 0.000,C 90.000,E1 281.827} C_DIS
LIN {X 0.234,Y -449.307,Z 1431.563,A 0.000,B 0.000,C 90.000,E1 281.299} C_DIS
LIN {X 0.195,Y -449.969,Z 1431.560,A 0.000,B 0.000,C 90.000,E1 280.782} C_DIS
LIN {X -0.194,Y -450.157,Z 1431.557,A 0.000,B 0.000,C 90.000,E1 280.310} C_DIS
LIN {X -0.141,Y -449.856,Z 1431.554,A 0.000,B 0.000,C 90.000,E1 279.782} C_DIS
LIN {X -0.162,Y -449.053,Z 1431.551,A 0.000,B 0.000,C 90.000,E1 279.265} C_DIS
LIN {X -0.181,Y -447.686,Z 1431.548,A 0.000,B 0.000,C 90.000,E1 278.746} C_DIS
LIN {X -0.138,Y -445.684,Z 1431.546,A 0.000,B 0.000,C 90.000,E1 278.219} C_DIS
LIN {X -0.167,Y -442.963,Z 1431.543,A 0.000,B 0.000,C 90.000,E1 277.701} C_DIS
LIN {X -0.212,Y -439.362,Z 1431.540,A 0.000,B 0.000,C 90.000,E1 277.182} C_DIS
LIN {X 0.001,Y -437.226,Z 1431.538,A 0.000,B 0.000,C 90.000,E1 276.891} C_DIS
LIN {X -0.073,Y -431.995,Z 1431.535,A 0.000,B 0.000,C 90.000,E1 276.372} C_DIS
LIN {X 0.113,Y -425.941,Z 1431.533,A 0.000,B 0.000,C 90.000,E1 275.853} C_DIS
LIN {X -0.103,Y -419.637,Z 1431.530,A 0.000,B 0.000,C 90.000,E1 275.454} C_DIS
LIN {X 0.145,Y -413.144,Z 1431.528,A 0.000,B 0.000,C 90.000,E1 275.049} C_DIS
LIN {X 0.003,Y -403.235,Z 1431.526,A 0.000,B 0.000,C 90.000,E1 274.588} C_DIS
LIN {X -0.041,Y -393.561,Z 1431.523,A 0.000,B 0.000,C 90.000,E1 274.188} C_DIS
LIN {X 0.173,Y -380.809,Z 1431.521,A 0.000,B 0.000,C 90.000,E1 273.669} C_DIS
LIN {X -0.168,Y -367.765,Z 1431.518,A 0.000,B 0.000,C 90.000,E1 273.269} C_DIS
LIN {X 0.089,Y -357.480,Z 1431.516,A 0.000,B 0.000,C 90.000,E1 272.922} C_DIS
LIN {X -0.099,Y -346.344,Z 1431.515,A 0.000,B 0.000,C 90.000,E1 272.694} C_DIS
LIN {X 0.072,Y -339.001,Z 1431.514,A 0.000,B 0.000,C 90.000,E1 272.522} C_DIS
LIN {X 0.049,Y -326.341,Z 1431.513,A 0.000,B 0.000,C 90.000,E1 272.350} C_DIS
LIN {X 0.152,Y -314.275,Z 1431.513,A 0.000,B 0.000,C 90.000,E1 272.236} C_DIS
LIN {X 0.005,Y -307.328,Z 1431.512,A 0.000,B 0.000,C 90.000,E1 272.236} C_DIS
LIN {X -0.025,Y -181.226,Z 1431.512,A 0.000,B 0.000,C 90.000,E1 272.236} C_DIS
LIN {X -0.026,Y -181.564,Z 1431.503,A 0.000,B 0.000,C 90.000,E1 270.516} C_DIS
LIN {X -0.036,Y -181.121,Z 1431.489,A 0.000,B 0.000,C 90.000,E1 267.993} C_DIS
LIN {X -0.047,Y -180.907,Z 1431.475,A 0.000,B 0.000,C 90.000,E1 265.469} C_DIS
LIN {X 0.009,Y -180.730,Z 1431.470,A 0.000,B 0.000,C 90.000,E1 264.609} C_DIS
LIN {X -0.070,Y -178.819,Z 1431.442,A 0.000,B 0.000,C 90.000,E1 259.567} C_DIS
LIN {X 0.013,Y -175.863,Z 1431.414,A 0.000,B 0.000,C 90.000,E1 254.448} C_DIS
LIN {X 0.062,Y -173.831,Z 1431.399,A 0.000,B 0.000,C 90.000,E1 251.873} C_DIS
LIN {X -0.003,Y -171.498,Z 1431.380,A 0.000,B 0.000,C 90.000,E1 248.465} C_DIS
LIN {X -0.017,Y -167.726,Z 1431.356,A 0.000,B 0.000,C 90.000,E1 244.152} C_DIS
LIN {X 0.000,Y -166.421,Z 1431.347,A 0.000,B 0.000,C 90.000,E1 242.410} C_DIS
LIN {X -0.002,Y -163.142,Z 1431.327,A 0.000,B 0.000,C 90.000,E1 238.918} C_DIS
LIN {X -0.036,Y -161.097,Z 1431.313,A 0.000,B 0.000,C 90.000,E1 236.294} C_DIS
LIN {X -0.053,Y -157.825,Z 1431.293,A 0.000,B 0.000,C 90.000,E1 232.763} C_DIS
LIN {X 0.011,Y -155.858,Z 1431.278,A 0.000,B 0.000,C 90.000,E1 230.070} C_DIS
LIN {X 0.067,Y -152.108,Z 1431.253,A 0.000,B 0.000,C 90.000,E1 225.567} C_DIS
LIN {X -0.026,Y -150.359,Z 1431.238,A 0.000,B 0.000,C 90.000,E1 222.894} C_DIS
LIN {X 0.013,Y -147.094,Z 1431.213,A 0.000,B 0.000,C 90.000,E1 218.338} C_DIS
LIN {X 0.008,Y -145.665,Z 1431.198,A 0.000,B 0.000,C 90.000,E1 215.598} C_DIS
LIN {X 0.011,Y -143.048,Z 1431.172,A 0.000,B 0.000,C 90.000,E1 211.003} C_DIS
LIN {X 0.011,Y -141.671,Z 1431.152,A 0.000,B 0.000,C 90.000,E1 207.308} C_DIS
LIN {X 0.056,Y -139.453,Z 1431.116,A 0.000,B 0.000,C 90.000,E1 200.791} C_DIS
LIN {X -0.023,Y -139.186,Z 1431.105,A 0.000,B 0.000,C 90.000,E1 198.960} C_DIS
LIN {X -0.001,Y -138.322,Z 1431.053,A 0.000,B 0.000,C 90.000,E1 189.613} C_DIS
LIN {X 0.007,Y -139.460,Z 1431.007,A 0.000,B 0.000,C 90.000,E1 181.203} C_DIS
LIN {X -0.053,Y -141.016,Z 1430.976,A 0.000,B 0.000,C 90.000,E1 175.641} C_DIS
LIN {X 0.037,Y -142.770,Z 1430.955,A 0.000,B 0.000,C 90.000,E1 171.894} C_DIS
LIN {X -0.008,Y -145.180,Z 1430.929,A 0.000,B 0.000,C 90.000,E1 167.297} C_DIS
LIN {X 0.026,Y -147.802,Z 1430.909,A 0.000,B 0.000,C 90.000,E1 163.614} C_DIS
LIN {X -0.079,Y -150.488,Z 1430.889,A 0.000,B 0.000,C 90.000,E1 160.007} C_DIS
LIN {X -0.007,Y -153.944,Z 1430.869,A 0.000,B 0.000,C 90.000,E1 156.357} C_DIS
LIN {X 0.057,Y -157.355,Z 1430.849,A 0.000,B 0.000,C 90.000,E1 152.743} C_DIS
LIN {X -0.001,Y -161.552,Z 1430.829,A 0.000,B 0.000,C 90.000,E1 149.203} C_DIS
LIN {X 0.012,Y -165.750,Z 1430.809,A 0.000,B 0.000,C 90.000,E1 145.674} C_DIS
LIN {X -0.001,Y -170.704,Z 1430.790,A 0.000,B 0.000,C 90.000,E1 142.190} C_DIS
LIN {X -0.090,Y -175.578,Z 1430.771,A 0.000,B 0.000,C 90.000,E1 138.771} C_DIS
LIN {X 0.030,Y -181.195,Z 1430.752,A 0.000,B 0.000,C 90.000,E1 135.324} C_DIS
LIN {X 0.023,Y -186.657,Z 1430.733,A 0.000,B 0.000,C 90.000,E1 131.962} C_DIS
LIN {X -0.032,Y -191.261,Z 1430.719,A 0.000,B 0.000,C 90.000,E1 129.483} C_DIS
LIN {X 0.047,Y -197.083,Z 1430.701,A 0.000,B 0.000,C 90.000,E1 126.171} C_DIS
LIN {X -0.007,Y -200.148,Z 1430.693,A 0.000,B 0.000,C 90.000,E1 124.659} C_DIS
LIN {X -0.047,Y -311.331,Z 1430.693,A 0.000,B 0.000,C 90.000,E1 124.659} C_DIS
LIN {X 0.103,Y -312.788,Z 1430.692,A 0.000,B 0.000,C 90.000,E1 124.612} C_DIS
LIN {X 0.132,Y -315.194,Z 1430.692,A 0.000,B 0.000,C 90.000,E1 124.532} C_DIS
LIN {X 0.192,Y -318.522,Z 1430.691,A 0.000,B 0.000,C 90.000,E1 124.326} C_DIS
LIN {X 0.054,Y -322.146,Z 1430.689,A 0.000,B 0.000,C 90.000,E1 123.992} C_DIS
LIN {X -0.021,Y -325.647,Z 1430.686,A 0.000,B 0.000,C 90.000,E1 123.452} C_DIS
LIN {X -0.205,Y -327.052,Z 1430.684,A 0.000,B 0.000,C 90.000,E1 123.166} C_DIS
LIN {X -0.050,Y -338.849,Z 1430.667,A 0.000,B 0.000,C 90.000,E1 120.001} C_DIS
LIN {X 0.113,Y -350.864,Z 1430.651,A 0.000,B 0.000,C 90.000,E1 117.206} C_DIS
LIN {X -0.009,Y -364.336,Z 1430.636,A 0.000,B 0.000,C 90.000,E1 114.515} C_DIS
LIN {X 0.013,Y -377.634,Z 1430.623,A 0.000,B 0.000,C 90.000,E1 112.153} C_DIS
LIN {X 0.234,Y -392.268,Z 1430.610,A 0.000,B 0.000,C 90.000,E1 109.812} C_DIS
LIN {X 0.054,Y -408.343,Z 1430.598,A 0.000,B 0.000,C 90.000,E1 107.583} C_DIS
LIN {X 0.150,Y -425.969,Z 1430.585,A 0.000,B 0.000,C 90.000,E1 105.371} C_DIS
LIN {X 0.090,Y -445.215,Z 1430.574,A 0.000,B 0.000,C 90.000,E1 103.244} C_DIS
LIN {X 0.186,Y -465.339,Z 1430.563,A 0.000,B 0.000,C 90.000,E1 101.243} C_DIS
LIN {X -0.057,Y -485.979,Z 1430.552,A 0.000,B 0.000,C 90.000,E1 99.443} C_DIS
LIN {X 0.082,Y -488.089,Z 1430.551,A 0.000,B 0.000,C 90.000,E1 99.208} C_DIS
LIN {X -0.024,Y -489.877,Z 1430.550,A 0.000,B 0.000,C 90.000,E1 98.973} C_DIS
LIN {X -0.205,Y -491.216,Z 1430.548,A 0.000,B 0.000,C 90.000,E1 98.746} C_DIS
LIN {X 0.088,Y -492.879,Z 1430.546,A 0.000,B 0.000,C 90.000,E1 98.219} C_DIS
LIN {X -0.172,Y -493.455,Z 1430.543,A 0.000,B 0.000,C 90.000,E1 97.757} C_DIS
LIN {X 0.068,Y -493.040,Z 1430.540,A 0.000,B 0.000,C 90.000,E1 97.239} C_DIS
LIN {X -0.177,Y -491.574,Z 1430.537,A 0.000,B 0.000,C 90.000,E1 96.777} C_DIS
LIN {X 0.215,Y -490.367,Z 1430.536,A 0.000,B 0.000,C 90.000,E1 96.486} C_DIS
LIN {X -0.165,Y -475.639,Z 1430.524,A 0.000,B 0.000,C 90.000,E1 94.302} C_DIS
LIN {X -0.101,Y -467.833,Z 1430.517,A 0.000,B 0.000,C 90.000,E1 93.037} C_DIS
LIN {X -0.177,Y -459.494,Z 1430.510,A 0.000,B 0.000,C 90.000,E1 91.776} C_DIS
LIN {X -0.194,Y -446.029,Z 1430.498,A 0.000,B 0.000,C 90.000,E1 89.714} C_DIS
LIN {X 0.087,Y -431.655,Z 1430.485,A 0.000,B 0.000,C 90.000,E1 87.306} C_DIS
LIN {X -0.215,Y -420.381,Z 1430.475,A 0.000,B 0.000,C 90.000,E1 85.469} C_DIS
LIN {X 0.115,Y -409.070,Z 1430.464,A 0.000,B 0.000,C 90.000,E1 83.514} C_DIS
LIN {X -0.096,Y -397.714,Z 1430.453,A 0.000,B 0.000,C 90.000,E1 81.602} C_DIS
LIN {X -0.099,Y -384.422,Z 1430.441,A 0.000,B 0.000,C 90.000,E1 79.342} C_DIS
LIN {X 0.165,Y -371.319,Z 1430.428,A 0.000,B 0.000,C 90.000,E1 76.992} C_DIS
LIN {X 0.137,Y -360.019,Z 1430.416,A 0.000,B 0.000,C 90.000,E1 74.936} C_DIS
LIN {X 0.124,Y -350.295,Z 1430.406,A 0.000,B 0.000,C 90.000,E1 73.142} C_DIS
LIN {X -0.057,Y -338.782,Z 1430.395,A 0.000,B 0.000,C 90.000,E1 71.040} C_DIS
LIN {X 0.050,Y -327.315,Z 1430.383,A 0.000,B 0.000,C 90.000,E1 68.847} C_DIS
LIN {X 0.062,Y -311.537,Z 1430.365,A 0.000,B 0.000,C 90.000,E1 65.665} C_DIS
LIN {X -0.013,Y -298.582,Z 1430.349,A 0.000,B 0.000,C 90.000,E1 62.743} C_DIS
LIN {X -0.075,Y -284.403,Z 1430.328,A 0.000,B 0.000,C 90.000,E1 59.076} C_DIS
LIN {X -0.042,Y -272.709,Z 1430.309,A 0.000,B 0.000,C 90.000,E1 55.642} C_DIS
LIN {X -0.029,Y -263.874,Z 1430.294,A 0.000,B 0.000,C 90.000,E1 52.844} C_DIS
LIN {X 0.079,Y -254.508,Z 1430.276,A 0.000,B 0.000,C 90.000,E1 49.622} C_DIS
LIN {X -0.136,Y -244.981,Z 1430.256,A 0.000,B 0.000,C 90.000,E1 46.053} C_DIS
LIN {X 0.045,Y -236.275,Z 1430.235,A 0.000,B 0.000,C 90.000,E1 42.324} C_DIS
LIN {X -0.018,Y -228.414,Z 1430.214,A 0.000,B 0.000,C 90.000,E1 38.588} C_DIS
LIN {X 0.005,Y -221.437,Z 1430.193,A 0.000,B 0.000,C 90.000,E1 34.771} C_DIS
LIN {X -0.066,Y -215.270,Z 1430.172,A 0.000,B 0.000,C 90.000,E1 30.924} C_DIS
LIN {X -0.034,Y -209.887,Z 1430.150,A 0.000,B 0.000,C 90.000,E1 27.001} C_DIS
LIN {X 0.023,Y -205.406,Z 1430.128,A 0.000,B 0.000,C 90.000,E1 23.025} C_DIS
LIN {X -0.012,Y -201.129,Z 1430.101,A 0.000,B 0.000,C 90.000,E1 18.236} C_DIS
LIN {X -0.040,Y -197.447,Z 1430.070,A 0.000,B 0.000,C 90.000,E1 12.591} C_DIS
LIN {X 0.000,Y -195.306,Z 1430.043,A 0.000,B 0.000,C 90.000,E1 7.701} C_DIS
LIN {X 0.022,Y -194.033,Z 1430.020,A 0.000,B 0.000,C 90.000,E1 3.612} C_DIS
LIN {X -0.094,Y -193.163,Z 1429.993,A 0.000,B 0.000,C 90.000,E1 358.740} C_DIS
LIN {X -0.024,Y -193.038,Z 1429.965,A 0.000,B 0.000,C 90.000,E1 353.799} C_DIS
LIN {X 0.011,Y -193.678,Z 1429.934,A 0.000,B 0.000,C 90.000,E1 348.049} C_DIS
LIN {X -0.001,Y -196.170,Z 1429.897,A 0.000,B 0.000,C 90.000,E1 341.511} C_DIS
LIN {X 0.068,Y -199.648,Z 1429.870,A 0.000,B 0.000,C 90.000,E1 336.613} C_DIS
LIN {X -0.058,Y -203.769,Z 1429.848,A 0.000,B 0.000,C 90.000,E1 332.615} C_DIS
LIN {X -0.038,Y -208.978,Z 1429.826,A 0.000,B 0.000,C 90.000,E1 328.614} C_DIS
LIN {X -0.103,Y -214.108,Z 1429.808,A 0.000,B 0.000,C 90.000,E1 325.468} C_DIS
LIN {X -0.014,Y -220.246,Z 1429.791,A 0.000,B 0.000,C 90.000,E1 322.316} C_DIS
LIN {X 0.030,Y -227.335,Z 1429.773,A 0.000,B 0.000,C 90.000,E1 319.218} C_DIS
LIN {X 0.007,Y -236.427,Z 1429.755,A 0.000,B 0.000,C 90.000,E1 315.810} C_DIS
LIN {X 0.085,Y -246.678,Z 1429.736,A 0.000,B 0.000,C 90.000,E1 312.447} C_DIS
LIN {X -0.019,Y -258.218,Z 1429.718,A 0.000,B 0.000,C 90.000,E1 309.197} C_DIS
LIN {X -0.150,Y -269.695,Z 1429.702,A 0.000,B 0.000,C 90.000,E1 306.377} C_DIS
LIN {X -0.033,Y -281.113,Z 1429.688,A 0.000,B 0.000,C 90.000,E1 303.913} C_DIS
LIN {X -0.052,Y -288.353,Z 1429.681,A 0.000,B 0.000,C 90.000,E1 302.546} C_DIS
LIN {X 0.019,Y -298.476,Z 1429.671,A 0.000,B 0.000,C 90.000,E1 300.846} C_DIS
LIN {X -0.087,Y -307.367,Z 1429.664,A 0.000,B 0.000,C 90.000,E1 299.539} C_DIS
LIN {X -0.079,Y -317.299,Z 1429.657,A 0.000,B 0.000,C 90.000,E1 298.231} C_DIS
LIN {X -0.174,Y -327.942,Z 1429.650,A 0.000,B 0.000,C 90.000,E1 297.001} C_DIS
LIN {X 0.008,Y -349.623,Z 1429.637,A 0.000,B 0.000,C 90.000,E1 294.695} C_DIS
LIN {X 0.002,Y -360.383,Z 1429.631,A 0.000,B 0.000,C 90.000,E1 293.590} C_DIS
LIN {X 0.131,Y -370.977,Z 1429.625,A 0.000,B 0.000,C 90.000,E1 292.461} C_DIS
LIN {X 0.007,Y -381.326,Z 1429.619,A 0.000,B 0.000,C 90.000,E1 291.354} C_DIS
LIN {X -0.053,Y -394.130,Z 1429.611,A 0.000,B 0.000,C 90.000,E1 289.939} C_DIS
LIN {X 0.145,Y -409.077,Z 1429.601,A 0.000,B 0.000,C 90.000,E1 288.236} C_DIS
LIN {X -0.061,Y -418.928,Z 1429.595,A 0.000,B 0.000,C 90.000,E1 287.166} C_DIS
LIN {X 0.180,Y -425.774,Z 1429.591,A 0.000,B 0.000,C 90.000,E1 286.315} C_DIS
LIN {X -0.174,Y -431.760,Z 1429.586,A 0.000,B 0.000,C 90.000,E1 285.552} C_DIS
LIN {X -0.123,Y -435.243,Z 1429.583,A 0.000,B 0.000,C 90.000,E1 285.009} C_DIS
LIN {X 0.038,Y -439.668,Z 1429.579,A 0.000,B 0.000,C 90.000,E1 284.189} C_DIS
LIN {X -0.083,Y -443.359,Z 1429.574,A 0.000,B 0.000,C 90.000,E1 283.411} C_DIS
LIN {X -0.071,Y -445.413,Z 1429.572,A 0.000,B 0.000,C 90.000,E1 282.883} C_DIS
LIN {X -0.046,Y -447.164,Z 1429.569,A 0.000,B 0.000,C 90.000,E1 282.355} C_DIS
LIN {X -0.015,Y -448.574,Z 1429.566,A 0.000,B 0.000,C 90.000,E1 281.827} C_DIS
LIN {X 0.025,Y -449.605,Z 1429.563,A 0.000,B 0.000,C 90.000,E1 281.299} C_DIS
LIN {X -0.011,Y -450.263,Z 1429.560,A 0.000,B 0.000,C 90.000,E1 280.782} C_DIS
LIN {X 0.044,Y -450.448,Z 1429.557,A 0.000,B 0.000,C 90.000,E1 280.254} C_DIS
LIN {X 0.099,Y -450.153,Z 1429.554,A 0.000,B 0.000,C 90.000,E1 279.726} C_DIS
LIN {X 0.080,Y -449.311,Z 1429.551,A 0.000,B 0.000,C 90.000,E1 279.208} C_DIS
LIN {X 0.130,Y -447.949,Z 1429.548,A 0.000,B 0.000,C 90.000,E1 278.681} C_DIS
LIN {X 0.107,Y -445.944,Z 1429.545,A 0.000,B 0.000,C 90.000,E1 278.163} C_DIS
LIN {X 0.078,Y -443.222,Z 1429.542,A 0.000,B 0.000,C 90.000,E1 277.644} C_DIS
LIN {X 0.033,Y -439.625,Z 1429.540,A 0.000,B 0.000,C 90.000,E1 277.125} C_DIS
LIN {X -0.188,Y -437.490,Z 1429.538,A 0.000,B 0.000,C 90.000,E1 276.891} C_DIS
LIN {X 0.180,Y -432.273,Z 1429.535,A 0.000,B 0.000,C 90.000,E1 276.315} C_DIS
LIN {X -0.049,Y -426.228,Z 1429.532,A 0.000,B 0.000,C 90.000,E1 275.853} C_DIS
LIN {X 0.195,Y -419.940,Z 1429.530,A 0.000,B 0.000,C 90.000,E1 275.391} C_DIS
LIN {X -0.028,Y -413.427,Z 1429.528,A 0.000,B 0.000,C 90.000,E1 275.049} C_DIS
LIN {X -0.160,Y -403.518,Z 1429.525,A 0.000,B 0.000,C 90.000,E1 274.588} C_DIS
LIN {X 0.180,Y -393.790,Z 1429.523,A 0.000,B 0.000,C 90.000,E1 274.131} C_DIS
LIN {X -0.018,Y -380.907,Z 1429.520,A 0.000,B 0.000,C 90.000,E1 273.669} C_DIS
LIN {X 0.033,Y -367.947,Z 1429.518,A 0.000,B 0.000,C 90.000,E1 273.212} C_DIS
LIN {X -0.033,Y -357.648,Z 1429.516,A 0.000,B 0.000,C 90.000,E1 272.922} C_DIS
LIN {X -0.159,Y -346.820,Z 1429.515,A 0.000,B 0.000,C 90.000,E1 272.694} C_DIS
LIN {X -0.039,Y -335.011,Z 1429.514,A 0.000,B 0.000,C 90.000,E1 272.465} C_DIS
LIN {X -0.017,Y -326.422,Z 1429.513,A 0.000,B 0.000,C 90.000,E1 272.350} C_DIS
LIN {X -0.094,Y -317.869,Z 1429.513,A 0.000,B 0.000,C 90.000,E1 272.293} C_DIS
LIN {X -0.003,Y -307.972,Z 1429.512,A 0.000,B 0.000,C 90.000,E1 272.236} C_DIS
LIN {X -0.029,Y -181.226,Z 1429.512,A 0.000,B 0.000,C 90.000,E1 272.236} C_DIS
LIN {X -0.052,Y -181.565,Z 1429.503,A 0.000,B 0.000,C 90.000,E1 270.516} C_DIS
LIN {X -0.062,Y -181.120,Z 1429.489,A 0.000,B 0.000,C 90.000,E1 267.993} C_DIS
LIN {X -0.073,Y -180.906,Z 1429.475,A 0.000,B 0.000,C 90.000,E1 265.469} C_DIS
LIN {X -0.016,Y -180.726,Z 1429.470,A 0.000,B 0.000,C 90.000,E1 264.609} C_DIS
LIN {X 0.081,Y -178.814,Z 1429.442,A 0.000,B 0.000,C 90.000,E1 259.511} C_DIS
LIN {X -0.012,Y -175.860,Z 1429.414,A 0.000,B 0.000,C 90.000,E1 254.448} C_DIS
LIN {X 0.036,Y -173.825,Z 1429.399,A 0.000,B 0.000,C 90.000,E1 251.873} C_DIS
LIN {X -0.028,Y -171.491,Z 1429.380,A 0.000,B 0.000,C 90.000,E1 248.465} C_DIS
LIN {X -0.041,Y -167.720,Z 1429.356,A 0.000,B 0.000,C 90.000,E1 244.152} C_DIS
LIN {X -0.024,Y -166.412,Z 1429.347,A 0.000,B 0.000,C 90.000,E1 242.410} C_DIS
LIN {X -0.026,Y -163.136,Z 1429.327,A 0.000,B 0.000,C 90.000,E1 238.918} C_DIS
LIN {X -0.060,Y -161.088,Z 1429.313,A 0.000,B 0.000,C 90.000,E1 236.294} C_DIS
LIN {X -0.077,Y -157.818,Z 1429.293,A 0.000,B 0.000,C 90.000,E1 232.763} C_DIS
LIN {X -0.012,Y -155.853,Z 1429.278,A 0.000,B 0.000,C 90.000,E1 230.070} C_DIS
LIN {X 0.043,Y -152.102,Z 1429.253,A 0.000,B 0.000,C 90.000,E1 225.567} C_DIS
LIN {X 0.062,Y -150.353,Z 1429.238,A 0.000,B 0.000,C 90.000,E1 222.852} C_DIS
LIN {X -0.009,Y -147.089,Z 1429.213,A 0.000,B 0.000,C 90.000,E1 218.338} C_DIS
LIN {X -0.014,Y -145.661,Z 1429.198,A 0.000,B 0.000,C 90.000,E1 215.598} C_DIS
LIN {X -0.011,Y -143.042,Z 1429.172,A 0.000,B 0.000,C 90.000,E1 211.003} C_DIS
LIN {X -0.011,Y -141.667,Z 1429.152,A 0.000,B 0.000,C 90.000,E1 207.308} C_DIS
LIN {X 0.033,Y -139.450,Z 1429.116,A 0.000,B 0.000,C 90.000,E1 200.791} C_DIS
LIN {X -0.045,Y -139.184,Z 1429.105,A 0.000,B 0.000,C 90.000,E1 198.960} C_DIS
LIN {X -0.022,Y -138.322,Z 1429.053,A 0.000,B 0.000,C 90.000,E1 189.613} C_DIS
LIN {X -0.015,Y -139.461,Z 1429.007,A 0.000,B 0.000,C 90.000,E1 181.203} C_DIS
LIN {X 0.065,Y -141.020,Z 1428.976,A 0.000,B 0.000,C 90.000,E1 175.584} C_DIS
LIN {X 0.020,Y -142.384,Z 1428.960,A 0.000,B 0.000,C 90.000,E1 172.818} C_DIS
LIN {X -0.059,Y -144.614,Z 1428.934,A 0.000,B 0.000,C 90.000,E1 168.229} C_DIS
LIN {X 0.003,Y -147.808,Z 1428.909,A 0.000,B 0.000,C 90.000,E1 163.614} C_DIS
LIN {X 0.039,Y -150.496,Z 1428.889,A 0.000,B 0.000,C 90.000,E1 159.953} C_DIS
LIN {X -0.030,Y -153.953,Z 1428.869,A 0.000,B 0.000,C 90.000,E1 156.357} C_DIS
LIN {X 0.032,Y -157.365,Z 1428.849,A 0.000,B 0.000,C 90.000,E1 152.743} C_DIS
LIN {X -0.024,Y -161.563,Z 1428.829,A 0.000,B 0.000,C 90.000,E1 149.203} C_DIS
LIN {X -0.012,Y -165.761,Z 1428.809,A 0.000,B 0.000,C 90.000,E1 145.674} C_DIS
LIN {X -0.026,Y -170.717,Z 1428.790,A 0.000,B 0.000,C 90.000,E1 142.190} C_DIS
LIN {X 0.017,Y -175.590,Z 1428.771,A 0.000,B 0.000,C 90.000,E1 138.728} C_DIS
LIN {X 0.004,Y -181.208,Z 1428.752,A 0.000,B 0.000,C 90.000,E1 135.324} C_DIS
LIN {X -0.004,Y -186.672,Z 1428.733,A 0.000,B 0.000,C 90.000,E1 131.962} C_DIS
LIN {X -0.060,Y -191.274,Z 1428.719,A 0.000,B 0.000,C 90.000,E1 129.483} C_DIS
LIN {X 0.020,Y -197.098,Z 1428.701,A 0.000,B 0.000,C 90.000,E1 126.171} C_DIS
LIN {X -0.052,Y -200.106,Z 1428.693,A 0.000,B 0.000,C 90.000,E1 124.692} C_DIS
LIN {X -0.117,Y -311.608,Z 1428.693,A 0.000,B 0.000,C 90.000,E1 124.692} C_DIS
LIN {X -0.045,Y -312.840,Z 1428.693,A 0.000,B 0.000,C 90.000,E1 124.659} C_DIS
LIN {X 0.089,Y -315.771,Z 1428.692,A 0.000,B 0.000,C 90.000,E1 124.532} C_DIS
LIN {X 0.018,Y -319.099,Z 1428.691,A 0.000,B 0.000,C 90.000,E1 124.326} C_DIS
LIN {X 0.111,Y -322.756,Z 1428.688,A 0.000,B 0.000,C 90.000,E1 123.913} C_DIS
LIN {X 0.052,Y -324.669,Z 1428.687,A 0.000,B 0.000,C 90.000,E1 123.627} C_DIS
LIN {X -0.186,Y -326.169,Z 1428.685,A 0.000,B 0.000,C 90.000,E1 123.372} C_DIS
LIN {X -0.159,Y -329.670,Z 1428.680,A 0.000,B 0.000,C 90.000,E1 122.418} C_DIS
LIN {X -0.063,Y -340.523,Z 1428.664,A 0.000,B 0.000,C 90.000,E1 119.589} C_DIS
LIN {X -0.016,Y -352.744,Z 1428.649,A 0.000,B 0.000,C 90.000,E1 116.821} C_DIS
LIN {X -0.096,Y -366.446,Z 1428.634,A 0.000,B 0.000,C 90.000,E1 114.131} C_DIS
LIN {X -0.029,Y -379.960,Z 1428.621,A 0.000,B 0.000,C 90.000,E1 111.770} C_DIS
LIN {X 0.108,Y -394.828,Z 1428.608,A 0.000,B 0.000,C 90.000,E1 109.450} C_DIS
LIN {X -0.013,Y -411.154,Z 1428.596,A 0.000,B 0.000,C 90.000,E1 107.221} C_DIS
LIN {X 0.148,Y -429.052,Z 1428.583,A 0.000,B 0.000,C 90.000,E1 105.009} C_DIS
LIN {X 0.210,Y -448.521,Z 1428.572,A 0.000,B 0.000,C 90.000,E1 102.883} C_DIS
LIN {X -0.021,Y -468.739,Z 1428.561,A 0.000,B 0.000,C 90.000,E1 100.950} C_DIS
LIN {X -0.123,Y -486.710,Z 1428.552,A 0.000,B 0.000,C 90.000,E1 99.378} C_DIS
LIN {X -0.058,Y -488.603,Z 1428.551,A 0.000,B 0.000,C 90.000,E1 99.151} C_DIS
LIN {X -0.161,Y -490.230,Z 1428.549,A 0.000,B 0.000,C 90.000,E1 98.916} C_DIS
LIN {X 0.219,Y -491.445,Z 1428.548,A 0.000,B 0.000,C 90.000,E1 98.624} C_DIS
LIN {X -0.046,Y -492.916,Z 1428.545,A 0.000,B 0.000,C 90.000,E1 98.163} C_DIS
LIN {X 0.184,Y -493.328,Z 1428.543,A 0.000,B 0.000,C 90.000,E1 97.644} C_DIS
LIN {X -0.063,Y -492.751,Z 1428.540,A 0.000,B 0.000,C 90.000,E1 97.182} C_DIS
LIN {X 0.180,Y -491.094,Z 1428.537,A 0.000,B 0.000,C 90.000,E1 96.663} C_DIS
LIN {X 0.084,Y -489.767,Z 1428.536,A 0.000,B 0.000,C 90.000,E1 96.429} C_DIS
LIN {X -0.130,Y -476.564,Z 1428.525,A 0.000,B 0.000,C 90.000,E1 94.473} C_DIS
LIN {X -0.077,Y -468.777,Z 1428.518,A 0.000,B 0.000,C 90.000,E1 93.212} C_DIS
LIN {X 0.076,Y -462.179,Z 1428.512,A 0.000,B 0.000,C 90.000,E1 92.178} C_DIS
LIN {X -0.118,Y -447.009,Z 1428.499,A 0.000,B 0.000,C 90.000,E1 89.885} C_DIS
LIN {X -0.090,Y -431.052,Z 1428.485,A 0.000,B 0.000,C 90.000,E1 87.249} C_DIS
LIN {X 0.020,Y -419.798,Z 1428.474,A 0.000,B 0.000,C 90.000,E1 85.355} C_DIS
LIN {X -0.032,Y -408.521,Z 1428.464,A 0.000,B 0.000,C 90.000,E1 83.451} C_DIS
LIN {X 0.096,Y -397.154,Z 1428.453,A 0.000,B 0.000,C 90.000,E1 81.489} C_DIS
LIN {X 0.141,Y -383.906,Z 1428.440,A 0.000,B 0.000,C 90.000,E1 79.218} C_DIS
LIN {X -0.052,Y -370.838,Z 1428.427,A 0.000,B 0.000,C 90.000,E1 76.937} C_DIS
LIN {X -0.028,Y -357.909,Z 1428.414,A 0.000,B 0.000,C 90.000,E1 74.574} C_DIS
LIN {X -0.072,Y -348.139,Z 1428.404,A 0.000,B 0.000,C 90.000,E1 72.779} C_DIS
LIN {X 0.137,Y -338.273,Z 1428.394,A 0.000,B 0.000,C 90.000,E1 70.913} C_DIS
LIN {X -0.105,Y -325.174,Z 1428.380,A 0.000,B 0.000,C 90.000,E1 68.465} C_DIS
LIN {X 0.052,Y -308.023,Z 1428.361,A 0.000,B 0.000,C 90.000,E1 64.921} C_DIS
LIN {X 0.014,Y -294.097,Z 1428.342,A 0.000,B 0.000,C 90.000,E1 61.641} C_DIS
LIN {X -0.020,Y -281.599,Z 1428.324,A 0.000,B 0.000,C 90.000,E1 58.280} C_DIS
LIN {X 0.073,Y -270.147,Z 1428.305,A 0.000,B 0.000,C 90.000,E1 54.815} C_DIS
LIN {X 0.036,Y -260.390,Z 1428.287,A 0.000,B 0.000,C 90.000,E1 51.662} C_DIS
LIN {X 0.051,Y -250.380,Z 1428.267,A 0.000,B 0.000,C 90.000,E1 48.081} C_DIS
LIN {X 0.051,Y -241.225,Z 1428.247,A 0.000,B 0.000,C 90.000,E1 44.433} C_DIS
LIN {X -0.055,Y -232.914,Z 1428.226,A 0.000,B 0.000,C 90.000,E1 40.744} C_DIS
LIN {X 0.015,Y -225.406,Z 1428.205,A 0.000,B 0.000,C 90.000,E1 36.950} C_DIS
LIN {X 0.127,Y -218.831,Z 1428.184,A 0.000,B 0.000,C 90.000,E1 33.086} C_DIS
LIN {X 0.106,Y -213.006,Z 1428.162,A 0.000,B 0.000,C 90.000,E1 29.205} C_DIS
LIN {X 0.059,Y -208.049,Z 1428.141,A 0.000,B 0.000,C 90.000,E1 25.283} C_DIS
LIN {X -0.031,Y -203.932,Z 1428.119,A 0.000,B 0.000,C 90.000,E1 21.334} C_DIS
LIN {X 0.051,Y -200.101,Z 1428.092,A 0.000,B 0.000,C 90.000,E1 16.496} C_DIS
LIN {X 0.002,Y -197.228,Z 1428.065,A 0.000,B 0.000,C 90.000,E1 11.658} C_DIS
LIN {X 0.006,Y -195.289,Z 1428.038,A 0.000,B 0.000,C 90.000,E1 6.777} C_DIS
LIN {X -0.046,Y -193.931,Z 1428.010,A 0.000,B 0.000,C 90.000,E1 1.892} C_DIS
LIN {X -0.012,Y -193.324,Z 1427.984,A 0.000,B 0.000,C 90.000,E1 357.078} C_DIS
LIN {X -0.043,Y -193.335,Z 1427.961,A 0.000,B 0.000,C 90.000,E1 352.989} C_DIS
LIN {X 0.042,Y -194.100,Z 1427.929,A 0.000,B 0.000,C 90.000,E1 347.229} C_DIS
LIN {X -0.086,Y -196.878,Z 1427.893,A 0.000,B 0.000,C 90.000,E1 340.732} C_DIS
LIN {X -0.030,Y -200.611,Z 1427.866,A 0.000,B 0.000,C 90.000,E1 335.845} C_DIS
LIN {X -0.027,Y -204.919,Z 1427.843,A 0.000,B 0.000,C 90.000,E1 331.820} C_DIS
LIN {X -0.036,Y -210.363,Z 1427.821,A 0.000,B 0.000,C 90.000,E1 327.837} C_DIS
LIN {X -0.058,Y -215.744,Z 1427.804,A 0.000,B 0.000,C 90.000,E1 324.689} C_DIS
LIN {X 0.076,Y -222.100,Z 1427.786,A 0.000,B 0.000,C 90.000,E1 321.537} C_DIS
LIN {X -0.011,Y -229.432,Z 1427.769,A 0.000,B 0.000,C 90.000,E1 318.485} C_DIS
LIN {X 0.024,Y -238.736,Z 1427.750,A 0.000,B 0.000,C 90.000,E1 315.081} C_DIS
LIN {X 0.001,Y -249.275,Z 1427.732,A 0.000,B 0.000,C 90.000,E1 311.757} C_DIS
LIN {X 0.130,Y -259.704,Z 1427.716,A 0.000,B 0.000,C 90.000,E1 308.830} C_DIS
LIN {X -0.027,Y -269.796,Z 1427.702,A 0.000,B 0.000,C 90.000,E1 306.377} C_DIS
LIN {X 0.097,Y -281.169,Z 1427.688,A 0.000,B 0.000,C 90.000,E1 303.913} C_DIS
LIN {X 0.082,Y -288.403,Z 1427.681,A 0.000,B 0.000,C 90.000,E1 302.546} C_DIS
LIN {X 0.005,Y -298.510,Z 1427.672,A 0.000,B 0.000,C 90.000,E1 300.875} C_DIS
LIN {X 0.056,Y -307.384,Z 1427.664,A 0.000,B 0.000,C 90.000,E1 299.539} C_DIS
LIN {X 0.069,Y -317.273,Z 1427.657,A 0.000,B 0.000,C 90.000,E1 298.231} C_DIS
LIN {X 0.026,Y -327.868,Z 1427.650,A 0.000,B 0.000,C 90.000,E1 297.001} C_DIS
LIN {X 0.023,Y -349.571,Z 1427.637,A 0.000,B 0.000,C 90.000,E1 294.719} C_DIS
LIN {X -0.179,Y -360.368,Z 1427.631,A 0.000,B 0.000,C 90.000,E1 293.643} C_DIS
LIN {X -0.071,Y -370.913,Z 1427.625,A 0.000,B 0.000,C 90.000,E1 292.514} C_DIS
LIN {X -0.127,Y -381.148,Z 1427.619,A 0.000,B 0.000,C 90.000,E1 291.408} C_DIS
LIN {X 0.184,Y -393.920,Z 1427.611,A 0.000,B 0.000,C 90.000,E1 289.939} C_DIS
LIN {X -0.147,Y -408.908,Z 1427.602,A 0.000,B 0.000,C 90.000,E1 288.308} C_DIS
LIN {X -0.227,Y -418.778,Z 1427.595,A 0.000,B 0.000,C 90.000,E1 287.221} C_DIS
LIN {X -0.111,Y -425.681,Z 1427.591,A 0.000,B 0.000,C 90.000,E1 286.386} C_DIS
LIN {X 0.066,Y -431.705,Z 1427.586,A 0.000,B 0.000,C 90.000,E1 285.552} C_DIS
LIN {X -0.114,Y -436.792,Z 1427.582,A 0.000,B 0.000,C 90.000,E1 284.773} C_DIS
LIN {X 0.058,Y -441.034,Z 1427.578,A 0.000,B 0.000,C 90.000,E1 283.953} C_DIS
LIN {X -0.049,Y -444.525,Z 1427.573,A 0.000,B 0.000,C 90.000,E1 283.175} C_DIS
LIN {X 0.201,Y -447.298,Z 1427.569,A 0.000,B 0.000,C 90.000,E1 282.355} C_DIS
LIN {X 0.234,Y -448.750,Z 1427.566,A 0.000,B 0.000,C 90.000,E1 281.827} C_DIS
LIN {X -0.253,Y -449.832,Z 1427.563,A 0.000,B 0.000,C 90.000,E1 281.366} C_DIS
LIN {X -0.202,Y -450.507,Z 1427.560,A 0.000,B 0.000,C 90.000,E1 280.838} C_DIS
LIN {X -0.146,Y -450.759,Z 1427.557,A 0.000,B 0.000,C 90.000,E1 280.310} C_DIS
LIN {X -0.167,Y -450.511,Z 1427.554,A 0.000,B 0.000,C 90.000,E1 279.792} C_DIS
LIN {X -0.108,Y -449.738,Z 1427.551,A 0.000,B 0.000,C 90.000,E1 279.265} C_DIS
LIN {X -0.123,Y -448.401,Z 1427.548,A 0.000,B 0.000,C 90.000,E1 278.746} C_DIS
LIN {X -0.075,Y -446.453,Z 1427.546,A 0.000,B 0.000,C 90.000,E1 278.219} C_DIS
LIN {X -0.101,Y -443.832,Z 1427.543,A 0.000,B 0.000,C 90.000,E1 277.701} C_DIS
LIN {X -0.143,Y -440.347,Z 1427.540,A 0.000,B 0.000,C 90.000,E1 277.182} C_DIS
LIN {X 0.072,Y -438.242,Z 1427.538,A 0.000,B 0.000,C 90.000,E1 276.891} C_DIS
LIN {X 0.001,Y -433.178,Z 1427.535,A 0.000,B 0.000,C 90.000,E1 276.372} C_DIS
LIN {X 0.180,Y -427.232,Z 1427.533,A 0.000,B 0.000,C 90.000,E1 275.853} C_DIS
LIN {X -0.079,Y -420.919,Z 1427.530,A 0.000,B 0.000,C 90.000,E1 275.454} C_DIS
LIN {X 0.079,Y -414.396,Z 1427.528,A 0.000,B 0.000,C 90.000,E1 275.049} C_DIS
LIN {X 0.167,Y -407.790,Z 1427.526,A 0.000,B 0.000,C 90.000,E1 274.702} C_DIS
LIN {X -0.098,Y -397.872,Z 1427.524,A 0.000,B 0.000,C 90.000,E1 274.302} C_DIS
LIN {X 0.063,Y -388.295,Z 1427.522,A 0.000,B 0.000,C 90.000,E1 273.898} C_DIS
LIN {X -0.017,Y -375.456,Z 1427.519,A 0.000,B 0.000,C 90.000,E1 273.440} C_DIS
LIN {X 0.118,Y -365.531,Z 1427.517,A 0.000,B 0.000,C 90.000,E1 273.094} C_DIS
LIN {X 0.153,Y -355.167,Z 1427.516,A 0.000,B 0.000,C 90.000,E1 272.808} C_DIS
LIN {X 0.086,Y -344.236,Z 1427.514,A 0.000,B 0.000,C 90.000,E1 272.579} C_DIS
LIN {X -0.033,Y -332.051,Z 1427.513,A 0.000,B 0.000,C 90.000,E1 272.407} C_DIS
LIN {X -0.097,Y -318.846,Z 1427.513,A 0.000,B 0.000,C 90.000,E1 272.293} C_DIS
LIN {X -0.007,Y -309.361,Z 1427.512,A 0.000,B 0.000,C 90.000,E1 272.236} C_DIS
LIN {X -0.031,Y -181.227,Z 1427.512,A 0.000,B 0.000,C 90.000,E1 272.236} C_DIS
LIN {X -0.054,Y -181.565,Z 1427.503,A 0.000,B 0.000,C 90.000,E1 270.516} C_DIS
LIN {X -0.064,Y -181.120,Z 1427.489,A 0.000,B 0.000,C 90.000,E1 267.993} C_DIS
LIN {X -0.076,Y -180.906,Z 1427.475,A 0.000,B 0.000,C 90.000,E1 265.469} C_DIS
LIN {X -0.019,Y -180.725,Z 1427.470,A 0.000,B 0.000,C 90.000,E1 264.609} C_DIS
LIN {X 0.079,Y -178.814,Z 1427.442,A 0.000,B 0.000,C 90.000,E1 259.511} C_DIS
LIN {X -0.015,Y -175.859,Z 1427.414,A 0.000,B 0.000,C 90.000,E1 254.448} C_DIS
LIN {X 0.034,Y -173.824,Z 1427.399,A 0.000,B 0.000,C 90.000,E1 251.873} C_DIS
LIN {X -0.030,Y -171.491,Z 1427.380,A 0.000,B 0.000,C 90.000,E1 248.465} C_DIS
LIN {X -0.043,Y -167.719,Z 1427.356,A 0.000,B 0.000,C 90.000,E1 244.152} C_DIS
LIN {X -0.027,Y -166.412,Z 1427.347,A 0.000,B 0.000,C 90.000,E1 242.410} C_DIS
LIN {X -0.028,Y -163.134,Z 1427.327,A 0.000,B 0.000,C 90.000,E1 238.918} C_DIS
LIN {X -0.063,Y -161.087,Z 1427.313,A 0.000,B 0.000,C 90.000,E1 236.294} C_DIS
LIN {X 0.047,Y -157.818,Z 1427.293,A 0.000,B 0.000,C 90.000,E1 232.718} C_DIS
LIN {X -0.015,Y -155.852,Z 1427.278,A 0.000,B 0.000,C 90.000,E1 230.070} C_DIS
LIN {X 0.041,Y -152.102,Z 1427.253,A 0.000,B 0.000,C 90.000,E1 225.567} C_DIS
LIN {X 0.059,Y -150.352,Z 1427.238,A 0.000,B 0.000,C 90.000,E1 222.852} C_DIS
LIN {X -0.011,Y -147.089,Z 1427.213,A 0.000,B 0.000,C 90.000,E1 218.338} C_DIS
LIN {X -0.017,Y -145.661,Z 1427.198,A 0.000,B 0.000,C 90.000,E1 215.598} C_DIS
LIN {X -0.014,Y -143.042,Z 1427.172,A 0.000,B 0.000,C 90.000,E1 211.003} C_DIS
LIN {X -0.013,Y -141.666,Z 1427.152,A 0.000,B 0.000,C 90.000,E1 207.308} C_DIS
LIN {X 0.032,Y -139.450,Z 1427.116,A 0.000,B 0.000,C 90.000,E1 200.791} C_DIS
LIN {X -0.047,Y -139.184,Z 1427.105,A 0.000,B 0.000,C 90.000,E1 198.960} C_DIS
LIN {X -0.024,Y -138.321,Z 1427.053,A 0.000,B 0.000,C 90.000,E1 189.613} C_DIS
LIN {X -0.017,Y -139.462,Z 1427.007,A 0.000,B 0.000,C 90.000,E1 181.203} C_DIS
LIN {X 0.063,Y -141.020,Z 1426.976,A 0.000,B 0.000,C 90.000,E1 175.584} C_DIS
LIN {X 0.018,Y -142.384,Z 1426.960,A 0.000,B 0.000,C 90.000,E1 172.818} C_DIS
LIN {X -0.061,Y -144.614,Z 1426.934,A 0.000,B 0.000,C 90.000,E1 168.229} C_DIS
LIN {X 0.001,Y -147.809,Z 1426.909,A 0.000,B 0.000,C 90.000,E1 163.614} C_DIS
LIN {X 0.088,Y -150.497,Z 1426.889,A 0.000,B 0.000,C 90.000,E1 159.934} C_DIS
LIN {X -0.032,Y -153.954,Z 1426.869,A 0.000,B 0.000,C 90.000,E1 156.357} C_DIS
LIN {X 0.031,Y -157.365,Z 1426.849,A 0.000,B 0.000,C 90.000,E1 152.743} C_DIS
LIN {X -0.027,Y -161.564,Z 1426.829,A 0.000,B 0.000,C 90.000,E1 149.203} C_DIS
LIN {X -0.015,Y -165.762,Z 1426.809,A 0.000,B 0.000,C 90.000,E1 145.674} C_DIS
LIN {X -0.029,Y -170.719,Z 1426.790,A 0.000,B 0.000,C 90.000,E1 142.190} C_DIS
LIN {X 0.014,Y -175.592,Z 1426.771,A 0.000,B 0.000,C 90.000,E1 138.728} C_DIS
LIN {X 0.002,Y -181.209,Z 1426.752,A 0.000,B 0.000,C 90.000,E1 135.324} C_DIS
LIN {X -0.006,Y -186.672,Z 1426.733,A 0.000,B 0.000,C 90.000,E1 131.962} C_DIS
LIN {X -0.062,Y -191.276,Z 1426.719,A 0.000,B 0.000,C 90.000,E1 129.483} C_DIS
LIN {X 0.018,Y -197.100,Z 1426.701,A 0.000,B 0.000,C 90.000,E1 126.171} C_DIS
LIN {X 0.040,Y -200.052,Z 1426.693,A 0.000,B 0.000,C 90.000,E1 124.692} C_DIS
LIN {X 0.027,Y -311.127,Z 1426.693,A 0.000,B 0.000,C 90.000,E1 124.692} C_DIS
LIN {X -0.080,Y -312.584,Z 1426.693,A 0.000,B 0.000,C 90.000,E1 124.692} C_DIS
LIN {X 0.085,Y -316.135,Z 1426.692,A 0.000,B 0.000,C 90.000,E1 124.532} C_DIS
LIN {X -0.037,Y -319.377,Z 1426.691,A 0.000,B 0.000,C 90.000,E1 124.326} C_DIS
LIN {X -0.077,Y -323.059,Z 1426.688,A 0.000,B 0.000,C 90.000,E1 123.913} C_DIS
LIN {X 0.071,Y -324.942,Z 1426.687,A 0.000,B 0.000,C 90.000,E1 123.579} C_DIS
LIN {X -0.052,Y -326.412,Z 1426.685,A 0.000,B 0.000,C 90.000,E1 123.293} C_DIS
LIN {X 0.064,Y -339.450,Z 1426.666,A 0.000,B 0.000,C 90.000,E1 119.823} C_DIS
LIN {X -0.055,Y -351.544,Z 1426.650,A 0.000,B 0.000,C 90.000,E1 117.078} C_DIS
LIN {X 0.169,Y -365.102,Z 1426.635,A 0.000,B 0.000,C 90.000,E1 114.335} C_DIS
LIN {X -0.130,Y -378.481,Z 1426.622,A 0.000,B 0.000,C 90.000,E1 112.025} C_DIS
LIN {X -0.029,Y -393.205,Z 1426.609,A 0.000,B 0.000,C 90.000,E1 109.704} C_DIS
LIN {X -0.063,Y -409.375,Z 1426.597,A 0.000,B 0.000,C 90.000,E1 107.457} C_DIS
LIN {X 0.048,Y -427.105,Z 1426.585,A 0.000,B 0.000,C 90.000,E1 105.245} C_DIS
LIN {X 0.026,Y -446.434,Z 1426.573,A 0.000,B 0.000,C 90.000,E1 103.119} C_DIS
LIN {X 0.106,Y -466.593,Z 1426.562,A 0.000,B 0.000,C 90.000,E1 101.130} C_DIS
LIN {X -0.122,Y -484.684,Z 1426.553,A 0.000,B 0.000,C 90.000,E1 99.557} C_DIS
LIN {X 0.026,Y -487.031,Z 1426.552,A 0.000,B 0.000,C 90.000,E1 99.321} C_DIS
LIN {X 0.096,Y -488.808,Z 1426.551,A 0.000,B 0.000,C 90.000,E1 99.095} C_DIS
LIN {X -0.006,Y -490.343,Z 1426.549,A 0.000,B 0.000,C 90.000,E1 98.859} C_DIS
LIN {X -0.111,Y -491.488,Z 1426.548,A 0.000,B 0.000,C 90.000,E1 98.624} C_DIS
LIN {X 0.112,Y -492.850,Z 1426.545,A 0.000,B 0.000,C 90.000,E1 98.106} C_DIS
LIN {X -0.144,Y -493.168,Z 1426.542,A 0.000,B 0.000,C 90.000,E1 97.644} C_DIS
LIN {X 0.096,Y -492.495,Z 1426.540,A 0.000,B 0.000,C 90.000,E1 97.125} C_DIS
LIN {X -0.149,Y -490.722,Z 1426.537,A 0.000,B 0.000,C 90.000,E1 96.663} C_DIS
LIN {X 0.241,Y -489.318,Z 1426.536,A 0.000,B 0.000,C 90.000,E1 96.372} C_DIS
LIN {X 0.015,Y -476.139,Z 1426.525,A 0.000,B 0.000,C 90.000,E1 94.416} C_DIS
LIN {X 0.061,Y -468.330,Z 1426.518,A 0.000,B 0.000,C 90.000,E1 93.154} C_DIS
LIN {X -0.005,Y -459.985,Z 1426.510,A 0.000,B 0.000,C 90.000,E1 91.892} C_DIS
LIN {X -0.053,Y -443.302,Z 1426.496,A 0.000,B 0.000,C 90.000,E1 89.312} C_DIS
LIN {X -0.139,Y -432.256,Z 1426.486,A 0.000,B 0.000,C 90.000,E1 87.478} C_DIS
LIN {X -0.005,Y -421.055,Z 1426.475,A 0.000,B 0.000,C 90.000,E1 85.584} C_DIS
LIN {X 0.045,Y -408.176,Z 1426.463,A 0.000,B 0.000,C 90.000,E1 83.394} C_DIS
LIN {X 0.161,Y -396.825,Z 1426.453,A 0.000,B 0.000,C 90.000,E1 81.432} C_DIS
LIN {X 0.148,Y -385.244,Z 1426.442,A 0.000,B 0.000,C 90.000,E1 79.454} C_DIS
LIN {X -0.021,Y -373.816,Z 1426.430,A 0.000,B 0.000,C 90.000,E1 77.465} C_DIS
LIN {X 0.076,Y -360.865,Z 1426.417,A 0.000,B 0.000,C 90.000,E1 75.102} C_DIS
LIN {X -0.014,Y -351.139,Z 1426.407,A 0.000,B 0.000,C 90.000,E1 73.323} C_DIS
LIN {X -0.075,Y -341.293,Z 1426.397,A 0.000,B 0.000,C 90.000,E1 71.511} C_DIS
LIN {X -0.042,Y -328.106,Z 1426.383,A 0.000,B 0.000,C 90.000,E1 69.028} C_DIS
LIN {X -0.001,Y -312.235,Z 1426.366,A 0.000,B 0.000,C 90.000,E1 65.845} C_DIS
LIN {X -0.052,Y -299.198,Z 1426.349,A 0.000,B 0.000,C 90.000,E1 62.922} C_DIS
LIN {X -0.060,Y -286.196,Z 1426.331,A 0.000,B 0.000,C 90.000,E1 59.587} C_DIS
LIN {X -0.040,Y -274.423,Z 1426.312,A 0.000,B 0.000,C 90.000,E1 56.167} C_DIS
LIN {X 0.082,Y -264.511,Z 1426.295,A 0.000,B 0.000,C 90.000,E1 53.004} C_DIS
LIN {X 0.051,Y -254.197,Z 1426.275,A 0.000,B 0.000,C 90.000,E1 49.461} C_DIS
LIN {X 0.005,Y -244.716,Z 1426.255,A 0.000,B 0.000,C 90.000,E1 45.850} C_DIS
LIN {X 0.005,Y -236.088,Z 1426.234,A 0.000,B 0.000,C 90.000,E1 42.162} C_DIS
LIN {X 0.112,Y -228.281,Z 1426.213,A 0.000,B 0.000,C 90.000,E1 38.382} C_DIS
LIN {X -0.051,Y -221.393,Z 1426.192,A 0.000,B 0.000,C 90.000,E1 34.612} C_DIS
LIN {X 0.054,Y -215.306,Z 1426.171,A 0.000,B 0.000,C 90.000,E1 30.718} C_DIS
LIN {X -0.013,Y -210.004,Z 1426.149,A 0.000,B 0.000,C 90.000,E1 26.821} C_DIS
LIN {X 0.053,Y -205.615,Z 1426.127,A 0.000,B 0.000,C 90.000,E1 22.845} C_DIS
LIN {X 0.026,Y -201.460,Z 1426.100,A 0.000,B 0.000,C 90.000,E1 18.055} C_DIS
LIN {X -0.069,Y -198.357,Z 1426.073,A 0.000,B 0.000,C 90.000,E1 13.244} C_DIS
LIN {X 0.035,Y -195.844,Z 1426.042,A 0.000,B 0.000,C 90.000,E1 7.530} C_DIS
LIN {X 0.078,Y -194.576,Z 1426.019,A 0.000,B 0.000,C 90.000,E1 3.440} C_DIS
LIN {X -0.091,Y -193.755,Z 1425.993,A 0.000,B 0.000,C 90.000,E1 358.740} C_DIS
LIN {X 0.002,Y -193.577,Z 1425.966,A 0.000,B 0.000,C 90.000,E1 353.799} C_DIS
LIN {X 0.060,Y -194.188,Z 1425.934,A 0.000,B 0.000,C 90.000,E1 348.049} C_DIS
LIN {X 0.012,Y -196.642,Z 1425.897,A 0.000,B 0.000,C 90.000,E1 341.529} C_DIS
LIN {X -0.022,Y -200.087,Z 1425.870,A 0.000,B 0.000,C 90.000,E1 336.666} C_DIS
LIN {X 0.052,Y -204.200,Z 1425.848,A 0.000,B 0.000,C 90.000,E1 332.615} C_DIS
LIN {X -0.091,Y -209.354,Z 1425.826,A 0.000,B 0.000,C 90.000,E1 328.663} C_DIS
LIN {X 0.035,Y -214.512,Z 1425.808,A 0.000,B 0.000,C 90.000,E1 325.468} C_DIS
LIN {X 0.005,Y -220.611,Z 1425.791,A 0.000,B 0.000,C 90.000,E1 322.351} C_DIS
LIN {X 0.049,Y -227.670,Z 1425.774,A 0.000,B 0.000,C 90.000,E1 319.256} C_DIS
LIN {X -0.138,Y -236.746,Z 1425.755,A 0.000,B 0.000,C 90.000,E1 315.891} C_DIS
LIN {X -0.045,Y -245.778,Z 1425.738,A 0.000,B 0.000,C 90.000,E1 312.894} C_DIS
LIN {X 0.009,Y -257.102,Z 1425.720,A 0.000,B 0.000,C 90.000,E1 309.600} C_DIS
LIN {X 0.091,Y -269.898,Z 1425.702,A 0.000,B 0.000,C 90.000,E1 306.377} C_DIS
LIN {X -0.168,Y -281.239,Z 1425.689,A 0.000,B 0.000,C 90.000,E1 303.992} C_DIS
LIN {X -0.031,Y -288.464,Z 1425.681,A 0.000,B 0.000,C 90.000,E1 302.594} C_DIS
LIN {X -0.117,Y -298.554,Z 1425.672,A 0.000,B 0.000,C 90.000,E1 300.924} C_DIS
LIN {X -0.072,Y -307.410,Z 1425.664,A 0.000,B 0.000,C 90.000,E1 299.589} C_DIS
LIN {X -0.066,Y -317.275,Z 1425.657,A 0.000,B 0.000,C 90.000,E1 298.281} C_DIS
LIN {X 0.179,Y -327.862,Z 1425.650,A 0.000,B 0.000,C 90.000,E1 297.001} C_DIS
LIN {X -0.087,Y -349.419,Z 1425.638,A 0.000,B 0.000,C 90.000,E1 294.771} C_DIS
LIN {X 0.047,Y -360.214,Z 1425.631,A 0.000,B 0.000,C 90.000,E1 293.643} C_DIS
LIN {X 0.214,Y -370.641,Z 1425.625,A 0.000,B 0.000,C 90.000,E1 292.514} C_DIS
LIN {X 0.186,Y -380.839,Z 1425.619,A 0.000,B 0.000,C 90.000,E1 291.408} C_DIS
LIN {X 0.129,Y -393.607,Z 1425.611,A 0.000,B 0.000,C 90.000,E1 289.993} C_DIS
LIN {X -0.181,Y -408.555,Z 1425.602,A 0.000,B 0.000,C 90.000,E1 288.362} C_DIS
LIN {X 0.079,Y -418.540,Z 1425.596,A 0.000,B 0.000,C 90.000,E1 287.221} C_DIS
LIN {X -0.211,Y -425.456,Z 1425.591,A 0.000,B 0.000,C 90.000,E1 286.441} C_DIS
LIN {X -0.039,Y -431.561,Z 1425.587,A 0.000,B 0.000,C 90.000,E1 285.607} C_DIS
LIN {X 0.010,Y -435.121,Z 1425.584,A 0.000,B 0.000,C 90.000,E1 285.064} C_DIS
LIN {X 0.170,Y -439.674,Z 1425.579,A 0.000,B 0.000,C 90.000,E1 284.245} C_DIS
LIN {X -0.055,Y -443.448,Z 1425.575,A 0.000,B 0.000,C 90.000,E1 283.480} C_DIS
LIN {X 0.060,Y -445.599,Z 1425.572,A 0.000,B 0.000,C 90.000,E1 282.939} C_DIS
LIN {X 0.086,Y -447.417,Z 1425.569,A 0.000,B 0.000,C 90.000,E1 282.411} C_DIS
LIN {X 0.117,Y -448.908,Z 1425.566,A 0.000,B 0.000,C 90.000,E1 281.883} C_DIS
LIN {X 0.070,Y -450.046,Z 1425.563,A 0.000,B 0.000,C 90.000,E1 281.366} C_DIS
LIN {X 0.123,Y -450.760,Z 1425.560,A 0.000,B 0.000,C 90.000,E1 280.838} C_DIS
LIN {X 0.180,Y -451.056,Z 1425.557,A 0.000,B 0.000,C 90.000,E1 280.310} C_DIS
LIN {X 0.161,Y -450.862,Z 1425.555,A 0.000,B 0.000,C 90.000,E1 279.792} C_DIS
LIN {X 0.221,Y -450.144,Z 1425.552,A 0.000,B 0.000,C 90.000,E1 279.265} C_DIS
LIN {X -0.237,Y -448.898,Z 1425.549,A 0.000,B 0.000,C 90.000,E1 278.803} C_DIS
LIN {X -0.187,Y -447.041,Z 1425.546,A 0.000,B 0.000,C 90.000,E1 278.276} C_DIS
LIN {X -0.210,Y -444.468,Z 1425.543,A 0.000,B 0.000,C 90.000,E1 277.757} C_DIS
LIN {X 0.020,Y -442.946,Z 1425.542,A 0.000,B 0.000,C 90.000,E1 277.466} C_DIS
LIN {X -0.029,Y -439.020,Z 1425.539,A 0.000,B 0.000,C 90.000,E1 276.947} C_DIS
LIN {X -0.096,Y -434.144,Z 1425.536,A 0.000,B 0.000,C 90.000,E1 276.429} C_DIS
LIN {X 0.029,Y -428.290,Z 1425.533,A 0.000,B 0.000,C 90.000,E1 275.910} C_DIS
LIN {X 0.116,Y -421.964,Z 1425.530,A 0.000,B 0.000,C 90.000,E1 275.454} C_DIS
LIN {X -0.193,Y -415.455,Z 1425.528,A 0.000,B 0.000,C 90.000,E1 275.106} C_DIS
LIN {X -0.155,Y -408.801,Z 1425.526,A 0.000,B 0.000,C 90.000,E1 274.759} C_DIS
LIN {X 0.131,Y -402.250,Z 1425.525,A 0.000,B 0.000,C 90.000,E1 274.416} C_DIS
LIN {X 0.076,Y -389.296,Z 1425.522,A 0.000,B 0.000,C 90.000,E1 273.898} C_DIS
LIN {X 0.050,Y -376.681,Z 1425.519,A 0.000,B 0.000,C 90.000,E1 273.440} C_DIS
LIN {X 0.163,Y -366.745,Z 1425.517,A 0.000,B 0.000,C 90.000,E1 273.094} C_DIS
LIN {X 0.174,Y -356.408,Z 1425.516,A 0.000,B 0.000,C 90.000,E1 272.808} C_DIS
LIN {X 0.141,Y -345.742,Z 1425.514,A 0.000,B 0.000,C 90.000,E1 272.579} C_DIS
LIN {X 0.032,Y -333.857,Z 1425.513,A 0.000,B 0.000,C 90.000,E1 272.407} C_DIS
LIN {X -0.047,Y -321.181,Z 1425.513,A 0.000,B 0.000,C 90.000,E1 272.293} C_DIS
LIN {X -0.017,Y -310.537,Z 1425.512,A 0.000,B 0.000,C 90.000,E1 272.236} C_DIS
LIN {X -0.067,Y -305.607,Z 1425.512,A 0.000,B 0.000,C 90.000,E1 272.236} C_DIS
LIN {X -0.069,Y -181.228,Z 1425.512,A 0.000,B 0.000,C 90.000,E1 272.236} C_DIS
LIN {X -0.020,Y -181.578,Z 1425.501,A 0.000,B 0.000,C 90.000,E1 270.172} C_DIS
LIN {X -0.030,Y -180.884,Z 1425.473,A 0.000,B 0.000,C 90.000,E1 265.122} C_DIS
LIN {X 0.029,Y -179.004,Z 1425.445,A 0.000,B 0.000,C 90.000,E1 260.038} C_DIS
LIN {X -0.052,Y -178.608,Z 1425.440,A 0.000,B 0.000,C 90.000,E1 259.218} C_DIS
LIN {X 0.016,Y -175.660,Z 1425.412,A 0.000,B 0.000,C 90.000,E1 254.102} C_DIS
LIN {X 0.021,Y -172.377,Z 1425.388,A 0.000,B 0.000,C 90.000,E1 249.826} C_DIS
LIN {X 0.036,Y -171.174,Z 1425.378,A 0.000,B 0.000,C 90.000,E1 248.103} C_DIS
LIN {X 0.079,Y -167.470,Z 1425.354,A 0.000,B 0.000,C 90.000,E1 243.768} C_DIS
LIN {X 0.012,Y -166.866,Z 1425.350,A 0.000,B 0.000,C 90.000,E1 242.922} C_DIS
LIN {X 0.066,Y -162.170,Z 1425.320,A 0.000,B 0.000,C 90.000,E1 237.661} C_DIS
LIN {X -0.013,Y -160.733,Z 1425.311,A 0.000,B 0.000,C 90.000,E1 235.928} C_DIS
LIN {X -0.034,Y -157.535,Z 1425.291,A 0.000,B 0.000,C 90.000,E1 232.396} C_DIS
LIN {X 0.023,Y -155.562,Z 1425.276,A 0.000,B 0.000,C 90.000,E1 229.703} C_DIS
LIN {X -0.043,Y -151.851,Z 1425.251,A 0.000,B 0.000,C 90.000,E1 225.243} C_DIS
LIN {X -0.029,Y -150.072,Z 1425.236,A 0.000,B 0.000,C 90.000,E1 222.528} C_DIS
LIN {X 0.005,Y -146.878,Z 1425.211,A 0.000,B 0.000,C 90.000,E1 217.971} C_DIS
LIN {X -0.006,Y -145.463,Z 1425.196,A 0.000,B 0.000,C 90.000,E1 215.231} C_DIS
LIN {X -0.088,Y -142.879,Z 1425.170,A 0.000,B 0.000,C 90.000,E1 210.669} C_DIS
LIN {X 0.033,Y -141.496,Z 1425.150,A 0.000,B 0.000,C 90.000,E1 206.924} C_DIS
LIN {X 0.018,Y -139.386,Z 1425.114,A 0.000,B 0.000,C 90.000,E1 200.429} C_DIS
LIN {X 0.006,Y -138.843,Z 1425.098,A 0.000,B 0.000,C 90.000,E1 197.638} C_DIS
LIN {X -0.070,Y -138.354,Z 1425.057,A 0.000,B 0.000,C 90.000,E1 190.197} C_DIS
LIN {X 0.062,Y -139.519,Z 1425.005,A 0.000,B 0.000,C 90.000,E1 180.802} C_DIS
LIN {X 0.003,Y -141.177,Z 1424.974,A 0.000,B 0.000,C 90.000,E1 175.241} C_DIS
LIN {X -0.026,Y -142.556,Z 1424.958,A 0.000,B 0.000,C 90.000,E1 172.470} C_DIS
LIN {X 0.041,Y -144.835,Z 1424.932,A 0.000,B 0.000,C 90.000,E1 167.825} C_DIS
LIN {X 0.027,Y -147.458,Z 1424.912,A 0.000,B 0.000,C 90.000,E1 164.157} C_DIS
LIN {X 0.055,Y -150.041,Z 1424.892,A 0.000,B 0.000,C 90.000,E1 160.496} C_DIS
LIN {X -0.082,Y -153.382,Z 1424.872,A 0.000,B 0.000,C 90.000,E1 156.922} C_DIS
LIN {X -0.034,Y -155.914,Z 1424.857,A 0.000,B 0.000,C 90.000,E1 154.204} C_DIS
LIN {X 0.081,Y -159.777,Z 1424.837,A 0.000,B 0.000,C 90.000,E1 150.589} C_DIS
LIN {X -0.071,Y -162.018,Z 1424.827,A 0.000,B 0.000,C 90.000,E1 148.869} C_DIS
LIN {X 0.042,Y -166.212,Z 1424.807,A 0.000,B 0.000,C 90.000,E1 145.308} C_DIS
LIN {X 0.045,Y -171.227,Z 1424.788,A 0.000,B 0.000,C 90.000,E1 141.823} C_DIS
LIN {X -0.032,Y -176.113,Z 1424.769,A 0.000,B 0.000,C 90.000,E1 138.405} C_DIS
LIN {X 0.084,Y -180.377,Z 1424.755,A 0.000,B 0.000,C 90.000,E1 135.810} C_DIS
LIN {X 0.062,Y -185.786,Z 1424.736,A 0.000,B 0.000,C 90.000,E1 132.447} C_DIS
LIN {X -0.005,Y -190.402,Z 1424.722,A 0.000,B 0.000,C 90.000,E1 129.967} C_DIS
LIN {X 0.010,Y -197.727,Z 1424.699,A 0.000,B 0.000,C 90.000,E1 125.851} C_DIS
LIN {X -0.050,Y -200.007,Z 1424.693,A 0.000,B 0.000,C 90.000,E1 124.739} C_DIS
LIN {X -0.113,Y -311.278,Z 1424.693,A 0.000,B 0.000,C 90.000,E1 124.739} C_DIS
LIN {X -0.123,Y -313.711,Z 1424.693,A 0.000,B 0.000,C 90.000,E1 124.692} C_DIS
LIN {X -0.024,Y -317.970,Z 1424.691,A 0.000,B 0.000,C 90.000,E1 124.452} C_DIS
LIN {X 0.161,Y -320.469,Z 1424.690,A 0.000,B 0.000,C 90.000,E1 124.199} C_DIS
LIN {X 0.080,Y -324.247,Z 1424.687,A 0.000,B 0.000,C 90.000,E1 123.706} C_DIS
LIN {X 0.164,Y -325.897,Z 1424.686,A 0.000,B 0.000,C 90.000,E1 123.372} C_DIS
LIN {X 0.077,Y -328.292,Z 1424.682,A 0.000,B 0.000,C 90.000,E1 122.752} C_DIS
LIN {X -0.028,Y -338.971,Z 1424.666,A 0.000,B 0.000,C 90.000,E1 119.951} C_DIS
LIN {X 0.000,Y -351.005,Z 1424.651,A 0.000,B 0.000,C 90.000,E1 117.180} C_DIS
LIN {X 0.038,Y -364.505,Z 1424.636,A 0.000,B 0.000,C 90.000,E1 114.463} C_DIS
LIN {X 0.072,Y -377.825,Z 1424.623,A 0.000,B 0.000,C 90.000,E1 112.099} C_DIS
LIN {X -0.064,Y -392.485,Z 1424.610,A 0.000,B 0.000,C 90.000,E1 109.812} C_DIS
LIN {X -0.250,Y -408.588,Z 1424.598,A 0.000,B 0.000,C 90.000,E1 107.583} C_DIS
LIN {X -0.161,Y -426.245,Z 1424.585,A 0.000,B 0.000,C 90.000,E1 105.371} C_DIS
LIN {X -0.129,Y -445.524,Z 1424.573,A 0.000,B 0.000,C 90.000,E1 103.231} C_DIS
LIN {X -0.124,Y -465.661,Z 1424.562,A 0.000,B 0.000,C 90.000,E1 101.243} C_DIS
LIN {X 0.202,Y -486.228,Z 1424.552,A 0.000,B 0.000,C 90.000,E1 99.378} C_DIS
LIN {X 0.212,Y -488.215,Z 1424.551,A 0.000,B 0.000,C 90.000,E1 99.151} C_DIS
LIN {X -0.183,Y -489.732,Z 1424.550,A 0.000,B 0.000,C 90.000,E1 98.973} C_DIS
LIN {X 0.126,Y -490.996,Z 1424.548,A 0.000,B 0.000,C 90.000,E1 98.690} C_DIS
LIN {X 0.025,Y -491.920,Z 1424.547,A 0.000,B 0.000,C 90.000,E1 98.454} C_DIS
LIN {X -0.234,Y -492.918,Z 1424.544,A 0.000,B 0.000,C 90.000,E1 97.992} C_DIS
LIN {X 0.066,Y -492.909,Z 1424.542,A 0.000,B 0.000,C 90.000,E1 97.466} C_DIS
LIN {X -0.183,Y -491.894,Z 1424.539,A 0.000,B 0.000,C 90.000,E1 97.004} C_DIS
LIN {X 0.151,Y -490.963,Z 1424.537,A 0.000,B 0.000,C 90.000,E1 96.720} C_DIS
LIN {X 0.055,Y -489.691,Z 1424.536,A 0.000,B 0.000,C 90.000,E1 96.486} C_DIS
LIN {X 0.132,Y -474.980,Z 1424.524,A 0.000,B 0.000,C 90.000,E1 94.245} C_DIS
LIN {X 0.186,Y -467.130,Z 1424.517,A 0.000,B 0.000,C 90.000,E1 92.980} C_DIS
LIN {X -0.124,Y -457.016,Z 1424.508,A 0.000,B 0.000,C 90.000,E1 91.489} C_DIS
LIN {X 0.091,Y -437.378,Z 1424.491,A 0.000,B 0.000,C 90.000,E1 88.339} C_DIS
LIN {X 0.189,Y -427.933,Z 1424.482,A 0.000,B 0.000,C 90.000,E1 86.731} C_DIS
LIN {X 0.129,Y -418.321,Z 1424.473,A 0.000,B 0.000,C 90.000,E1 85.122} C_DIS
LIN {X 0.006,Y -407.074,Z 1424.462,A 0.000,B 0.000,C 90.000,E1 83.223} C_DIS
LIN {X 0.156,Y -395.744,Z 1424.452,A 0.000,B 0.000,C 90.000,E1 81.254} C_DIS
LIN {X 0.056,Y -384.191,Z 1424.441,A 0.000,B 0.000,C 90.000,E1 79.285} C_DIS
LIN {X -0.058,Y -372.767,Z 1424.429,A 0.000,B 0.000,C 90.000,E1 77.285} C_DIS
LIN {X -0.044,Y -361.433,Z 1424.418,A 0.000,B 0.000,C 90.000,E1 75.227} C_DIS
LIN {X -0.086,Y -350.090,Z 1424.406,A 0.000,B 0.000,C 90.000,E1 73.142} C_DIS
LIN {X 0.160,Y -340.218,Z 1424.396,A 0.000,B 0.000,C 90.000,E1 71.275} C_DIS
LIN {X -0.037,Y -327.043,Z 1424.382,A 0.000,B 0.000,C 90.000,E1 68.827} C_DIS
LIN {X 0.058,Y -309.690,Z 1424.363,A 0.000,B 0.000,C 90.000,E1 65.305} C_DIS
LIN {X 0.059,Y -296.910,Z 1424.347,A 0.000,B 0.000,C 90.000,E1 62.359} C_DIS
LIN {X 0.131,Y -285.384,Z 1424.330,A 0.000,B 0.000,C 90.000,E1 59.331} C_DIS
LIN {X 0.038,Y -273.691,Z 1424.311,A 0.000,B 0.000,C 90.000,E1 55.928} C_DIS
LIN {X 0.148,Y -263.855,Z 1424.293,A 0.000,B 0.000,C 90.000,E1 52.763} C_DIS
LIN {X 0.103,Y -253.635,Z 1424.274,A 0.000,B 0.000,C 90.000,E1 49.218} C_DIS
LIN {X -0.134,Y -244.216,Z 1424.253,A 0.000,B 0.000,C 90.000,E1 45.648} C_DIS
LIN {X 0.022,Y -235.664,Z 1424.233,A 0.000,B 0.000,C 90.000,E1 41.919} C_DIS
LIN {X -0.030,Y -227.927,Z 1424.212,A 0.000,B 0.000,C 90.000,E1 38.177} C_DIS
LIN {X 0.110,Y -221.109,Z 1424.191,A 0.000,B 0.000,C 90.000,E1 34.326} C_DIS
LIN {X 0.088,Y -215.089,Z 1424.169,A 0.000,B 0.000,C 90.000,E1 30.463} C_DIS
LIN {X 0.016,Y -209.874,Z 1424.148,A 0.000,B 0.000,C 90.000,E1 26.565} C_DIS
LIN {X 0.076,Y -205.572,Z 1424.126,A 0.000,B 0.000,C 90.000,E1 22.589} C_DIS
LIN {X -0.022,Y -201.516,Z 1424.099,A 0.000,B 0.000,C 90.000,E1 17.819} C_DIS
LIN {X -0.111,Y -198.512,Z 1424.072,A 0.000,B 0.000,C 90.000,E1 13.008} C_DIS
LIN {X -0.004,Y -196.058,Z 1424.041,A 0.000,B 0.000,C 90.000,E1 7.296} C_DIS
LIN {X -0.016,Y -194.630,Z 1424.013,A 0.000,B 0.000,C 90.000,E1 2.407} C_DIS
LIN {X 0.056,Y -193.989,Z 1423.988,A 0.000,B 0.000,C 90.000,E1 357.879} C_DIS
LIN {X -0.037,Y -193.876,Z 1423.961,A 0.000,B 0.000,C 90.000,E1 352.996} C_DIS
LIN {X 0.095,Y -194.625,Z 1423.929,A 0.000,B 0.000,C 90.000,E1 347.229} C_DIS
LIN {X -0.007,Y -197.362,Z 1423.893,A 0.000,B 0.000,C 90.000,E1 340.732} C_DIS
LIN {X -0.014,Y -201.040,Z 1423.866,A 0.000,B 0.000,C 90.000,E1 335.869} C_DIS
LIN {X -0.009,Y -205.352,Z 1423.844,A 0.000,B 0.000,C 90.000,E1 331.847} C_DIS
LIN {X -0.017,Y -210.755,Z 1423.821,A 0.000,B 0.000,C 90.000,E1 327.867} C_DIS
LIN {X 0.087,Y -216.140,Z 1423.804,A 0.000,B 0.000,C 90.000,E1 324.689} C_DIS
LIN {X -0.077,Y -222.469,Z 1423.787,A 0.000,B 0.000,C 90.000,E1 321.618} C_DIS
LIN {X -0.067,Y -230.753,Z 1423.767,A 0.000,B 0.000,C 90.000,E1 318.162} C_DIS
LIN {X 0.009,Y -240.158,Z 1423.749,A 0.000,B 0.000,C 90.000,E1 314.757} C_DIS
LIN {X 0.028,Y -250.791,Z 1423.730,A 0.000,B 0.000,C 90.000,E1 311.434} C_DIS
LIN {X 0.029,Y -261.329,Z 1423.714,A 0.000,B 0.000,C 90.000,E1 308.543} C_DIS
LIN {X -0.008,Y -269.986,Z 1423.702,A 0.000,B 0.000,C 90.000,E1 306.423} C_DIS
LIN {X -0.043,Y -281.313,Z 1423.689,A 0.000,B 0.000,C 90.000,E1 303.992} C_DIS
LIN {X -0.057,Y -288.522,Z 1423.681,A 0.000,B 0.000,C 90.000,E1 302.625} C_DIS
LIN {X 0.019,Y -298.596,Z 1423.672,A 0.000,B 0.000,C 90.000,E1 300.924} C_DIS
LIN {X -0.084,Y -307.449,Z 1423.664,A 0.000,B 0.000,C 90.000,E1 299.617} C_DIS
END
